    # this function converts a matrix to axis angle representations
    # this matrix is usually a resulting matrix (result of matrix multiplication) in normal use, given as a list
    # returns a list of [rx,ry,rz]
    def convert_matrix_to_axang(matrix1):
        # retrieve values
        a11 = matrix1[0]
        a12 = matrix1[1]
        a13 = matrix1[2]
        a21 = matrix1[3]
        a22 = matrix1[4]
        a23 = matrix1[5]
        a31 = matrix1[6]
        a32 = matrix1[7]
        a33 = matrix1[8]

        # First Half: find the angle
        # find the trace
        # using the formula: trace = a11 + a22 + a33
        trace = a11 + a22 + a33
        # find the angle using the formula: trace(matrix) = 1 + 2 cos(angle)
        angle = acos((trace - 1.0)/2.0)

        # Second Half: calculate the rotation axis
        axisxraw = a32 - a23
        axisyraw = a13 - a31
        axiszraw = a21 - a12
        # normalize axis
        magnitude = sqrt(axisxraw*axisxraw + axisyraw*axisyraw + axiszraw*axiszraw)
        axisxunit = axisxraw / magnitude
        axisyunit = axisyraw / magnitude
        axiszunit = axiszraw / magnitude

        # combine axis and angle into rxryrz representation
        rxout = axisxunit * angle
        ryout = axisyunit * angle
        rzout = axiszunit * angle
        return [rxout, ryout, rzout]
    end

    # this function takes a rotation and calculates the corresponding rotation matrix
    # input is (axis, direction, angle in radians)
    # example is ("x", 1, pi/6) = a 30 degree turn around the x axis in the positive direction (right hand rule)
    # returns a matrix (a list of 9 values)
    def get_rotation_matrix_from_description(axis, direction, angle):
        # get the angle
        a = angle * direction
        # get the axis
        if axis == "x" or axis == "X":
            matrix = [1, 0, 0, 0, cos(a), -1 * sin(a), 0, sin(a), cos(a)]
            return matrix
        end
        if axis == "y" or axis == "Y":
            matrix = [cos(a), 0, sin(a), 0, 1, 0, -1*sin(a), 0, cos(a)]
            return matrix
        end
        if axis == "z" or axis == "Z":
            matrix = [cos(a), -1*sin(a), 0, sin(a), cos(a), 0, 0, 0, 1]
            return matrix
        end
        # bad
        popuptext = "Error in get_rotation_matrix_from_description. "
        # infinite loop
        while 1==1:
          popup(popuptext, title="Code Error",blocking=True)
        end
    end

    def main_calculate_step_right(p11, p12, p21, p22, p3, p13, p23, noncappingsidewallthick, cappingsidewallthick, tcp_pose_top):
        struct1 = analyze_touchpoints_only(p11, p12, p21, p22, p3)
        list1 = analyze_vertical_touchpoints(p11, p12, p13, p21, p22, p23, p3)
        #struct2 = calculate_DOtA_points_right(struct1, list1, chamferover)
        #validity = check_validity_right(struct1, struct2)
        struct2 = calculate_DAaU_step_right(struct1, list1, noncappingsidewallthick, cappingsidewallthick, tcp_pose_top)
        return struct2
    end

    def main_calculate_step_left(p11, p12, p21, p22, p3, p13, p23, noncappingsidewallthick, cappingsidewallthick, tcp_pose_top):
        struct1 = analyze_touchpoints_only(p11, p12, p21, p22, p3)
        list1 = analyze_vertical_touchpoints(p11, p12, p13, p21, p22, p23, p3)
        #struct2 = calculate_DOtA_points_right(struct1, list1, chamferover)
        #validity = check_validity_right(struct1, struct2)
        struct2 = calculate_DAaU_step_left(struct1, list1, cappingsidewallthick, noncappingsidewallthick, tcp_pose_top)
        return struct2
    end

    # analyze_touchpoints_only()
    # it takes 5 arguments as points
    # it returns a struct containing: (pointintersect, heading1, heading2, heading3, l1delxunit, l1delyunit, l2delxunit, l2delyunit)
    #   FIND HEADINGS
    #for each heading, find the angle of the line with respect to the pos x axis. then add/subtract 90 degrees because you want to be perpendicular to that
    # so, heading1 finds the angle (from the +x axis) to the position pointing perpendicularly into the box.
    # we need to be +90 degrees of all 3 headings. (but we can ignore heading 2)
    def step_right_demo(struct1):
        pointintersect = struct1[0]
        x = pointintersect[0]
        y = pointintersect[1]
        z = pointintersect[2]
        heading1 = struct1[1]
        heading1adj1 = heading1 + pi/2 #(90 deg) (parrallel to edge not perpendicular into
        heading1adj2 = heading1adj1 - pi/2 #(90 deg) (from y+ not x+)
        # heading1 == heading1adj2. ok
        m1 = get_rotation_matrix_from_description("z", 1, heading1)
        # at this point we would multiply matrices, but there is only one matrix
        rxryrz = convert_matrix_to_axang(m1)
        point_demo = p[x, y, z, rxryrz[0], rxryrz[1], rxryrz[2]]
        popup(point_demo)
        movej(point_demo, a=1.4, v=0.1)
        popup(point_demo)
        ret = struct(point_demo = point_demo)
        return ret
    end

    # for a right step corner, calculate the toolpath points for a L (under) then Up and Around weld.
    def calculate_LtUA_step_right(struct1, list1, rightwallthick, leftwallthick, tcp_pose_top):
        # get the stuff from the struct
        pointintersect = struct1[0]
        heading1 = struct1[1]
        heading2 = struct1[2]
        heading3 = struct1[3]
        l1delxunit = struct1[4]
        l1delyunit = struct1[5]
        l2delxunit = struct1[6]
        l2delyunit = struct1[7]

        # FIND THE POINTS ON THE LINES OF THE FIRST TURN PATH
        # find locations 8 inches away from  intersect point
        # CONST
        welddistance1 = 3 # first path first leg
        welddistance2 = 3 # first path second leg
        welddistance3 = 8 # vertical weld distance

        # inches
        wd1 = welddistance1 * 25.4 / 1000
        wd2 = welddistance2 * 25.4 / 1000
        wd3 = welddistance3 * 25.4 / 1000
        leftwallthickmm = leftwallthick * 25.4 / 1000 # in this step corner right, this is distance from left edge
        rightwallthickmm =  rightwallthick * 25.4 / 1000 # in this step corner right, this is distance from right edge


        # weld distance is the distance that it will weld. this will make it start at the z height that the user specified
        #wd1 = tcp_pose_top[2] - pointintersect[2] - zup # this will need to change for step corner right

        # point bottom (point of intersection of the two chamfers on the bottom)
        xbottom = pointintersect[0] + l1delxunit * leftwallthickmm + l2delxunit * rightwallthickmm
        ybottom = pointintersect[1] + l1delyunit * leftwallthickmm + l2delyunit * rightwallthickmm
        z = pointintersect[2]

        # point 1
        x = xbottom + l1delxunit * wd1
        y = ybottom + l1delyunit * wd1

        m1 = get_rotation_matrix_from_description("z", 1, heading1)
        # at this point we would multiply matrices, but there is only one matrix
        rxryrz = convert_matrix_to_axang(m1)
        rx = rxryrz[0]
        ry = rxryrz[1]
        rz = rxryrz[2]
        point1 = p[x, y, z, rx, ry, rz]

        # point 2
        point2 = p[xbottom, ybottom, z, rx, ry, rz]

        # point 4
        m1 = get_rotation_matrix_from_description("z", 1, heading3)
        # at this point we would multiply matrices, but there is only one matrix
        rxryrz = convert_matrix_to_axang(m1)
        rx = rxryrz[0]
        ry = rxryrz[1]
        rz = rxryrz[2]
        point4 = p[xbottom, ybottom, z, rx, ry, rz]

        # point 5
        x = xbottom + l2delxunit * wd2
        y = ybottom + l2delyunit * wd2
        point5 = p[x, y, z, rx, ry, rz]


        # form struct
        struct2 = struct(point1=point1, point2=point2, point4=point4, point5=point5, point_1=point1, point_2=point1, point_3=point1, point_4=point1, point_5=point1)
        return struct2
    end

    # step corner with two seams on bottom face
    # vertical seam on left side of corner
    # Down Around and Under weld path, then Back Away
    # the first path uses backofhole TCP, the second path uses pretend_welder TCP
    def calculate_DAaU_step_left(struct1, listleans, rightwallthick, leftwallthick, tcp_pose_top):
        # get the stuff from the struct
        pointintersect = struct1[0]
        heading1 = struct1[1]
        heading2 = struct1[2]
        heading3 = struct1[3]
        l1delxunit = struct1[4]
        l1delyunit = struct1[5]
        l2delxunit = struct1[6]
        l2delyunit = struct1[7]

        # FIND THE POINTS ON THE LINES OF THE FIRST TURN PATH
        # find locations 8 inches away from  intersect point
        # CONST
        welddistance1 = 8 # first path first leg (down)
        welddistance2 = 3 # first path second leg (under) # inches
        welddistance3 = 3 # second path (back away) # inches

        wd1 = tcp_pose_top[2] - pointintersect[2] # the touchpoint minus the corner
        wd2 = welddistance2 * 25.4 / 1000
        wd3 = welddistance3 * 25.4 / 1000
        leftwallthickmm = leftwallthick * 25.4 / 1000 # in this step corner right, this is distance from left edge
        rightwallthickmm =  rightwallthick * 25.4 / 1000 # in this step corner right, this is distance from right edge

        # first, calculate the location of the bottom of the vertical chamfer (where point2 would be if there weren't any circle motion
        x = pointintersect[0] + l2delxunit * rightwallthickmm
        y = pointintersect[1] + l2delyunit * rightwallthickmm
        z = pointintersect[2]
        pointbottomvcham = p[x, y, z, 0, 0, 0]

        # calculate the rxryrz for facing the vertical chamfer, with the preheat down
        rxryrz = convert_heading_to_axang_preheatdown(heading3)
        rx = rxryrz[0]
        ry = rxryrz[1]
        rz = rxryrz[2]

        # next, calculate point1 using the listleans
        point1 = p[x + wd1*listleans[0], y + wd1*listleans[1], z + wd1, rx, ry, rz] # add in the listleans factor to follow the face of the box as we move up

        # calculate rxryrz for point2 and point2a (based on heading1). should be very similar to the heading for point1
        # only use the right side taps for circle move related things
        heading3basedh1 = heading1 - pi/2 # heading1 based on heading3
        rxryrz = convert_heading_to_axang_preheatdown(heading3basedh1)
        rx = rxryrz[0]
        ry = rxryrz[1]
        rz = rxryrz[2]

        # the round over distance is the distance from pointbottomvcham to point2 (which will be the same as distance to p4)
        roundoverdistance = 0.05
        rod = roundoverdistance * 25.4 / 1000
        point2 = p[x, y, z + rod, rx, ry, rz]

        # calculate point2a, which is directly above pointbottomvcham (used to straighten weldpath before circlemove)
        straightlength = 1.0 # the moveP blend radius for the circle move was set to 1.0 mm in FloorCorner. we should be more than 2.0mm away from point2
        sld = straightlength * 25.4 / 1000
        point2a = p[x, y, z + sld, rx, ry, rz]

        # calculate the rxryrz for facing the underneath section, with the preheat facing parallel to the right edge (rx and ry should be 0 because gun is facing up)
        # to convert heading1 into the description, subtract 90 degrees to go parallel  instead of into. subtract 90 degrees to start from y+ instead of x+
        heading1descr = heading1 - pi
        m1 = get_rotation_matrix_from_description("z", 1, heading1descr)
        rxryrz = convert_matrix_to_axang(m1)
        rx = rxryrz[0]
        ry = rxryrz[1]
        rz = rxryrz[2]

        # calculate point4
        p4x = x + l1delxunit * rod
        p4y = y + l1delyunit * rod
        point4 = p[p4x, p4y, z, rx, ry, rz]

        # calculate point5
        p5x = x + l1delxunit * wd2
        p5y = y + l1delyunit * wd2
        point5 = p[p5x, p5y, z, rx, ry, rz]

        # calculate point3
        # we know that the angle is exactly 90 degrees
        delta = calc_rod_midpoint_90deg(rod)
        p3z = z + delta
        p3x = x + delta * l1delxunit
        p3y = y + delta * l1delyunit

        # calculate rxryrz
        m1 = get_rotation_matrix_from_description("x", -1, 45 * pi / 180) # rotation 1: 45 degrees forward about x axis
        m2 = get_rotation_matrix_from_description("z", 1, heading1descr) # rotation 2
        m3 = multiply_matrix(m2, m1) #we rotate m1 first then m2, so we multiply in backwards order: 2 then 1
        rxryrz = convert_matrix_to_axang(m3)
        rx = rxryrz[0]
        ry = rxryrz[1]
        rz = rxryrz[2]
        point3 = p[p3x, p3y, p3z, rx, ry, rz]

        #todo: calculate trail out point

        # calculate back-away (points 201 and 202)
        pushtipforward = 0.006 # 6 millimeters forward. the tip needs to clear the capping wall's angled chamfer to not BONK when getting into position
        p201x = x + l1delxunit * leftwallthickmm + l2delxunit * pushtipforward
        p201y = y + l1delyunit * leftwallthickmm + l2delyunit * pushtipforward

        # calculate rxryrz
        m1 = get_rotation_matrix_from_description("z", 1, heading3)
        # minus pi/2 for the different start point. minus pi/2 for parallel not perpendicular into
        rxryrz = convert_matrix_to_axang(m1)
        rx = rxryrz[0]
        ry = rxryrz[1]
        rz = rxryrz[2]
        point201 = p[p201x, p201y, z, rx, ry, rz]

        # calculate point 202
        p202x = p201x + wd3 * l2delxunit
        p202y = p201y + wd3 * l2delyunit
        point202 = p[p202x, p202y, z, rx, ry, rz]

        struct2 = struct(point1=point1, point2a=point2a, point2=point2, point3=point3, point4=point4, point5=point5, point201=point201, point202=point202)
        return struct2
    end

    # step corner with two seams on bottom face
    # vertical seam on right side of corner
    # Down Around and Under weld path, then Back Away
    # the first path uses backofhole TCP, the second path uses pretend_welder TCP
    def calculate_DAaU_step_right(struct1, listleans, rightwallthick, leftwallthick, tcp_pose_top):
        # get the stuff from the struct
        pointintersect = struct1[0]
        heading1 = struct1[1]
        heading2 = struct1[2]
        heading3 = struct1[3]
        l1delxunit = struct1[4]
        l1delyunit = struct1[5]
        l2delxunit = struct1[6]
        l2delyunit = struct1[7]

        # FIND THE POINTS ON THE LINES OF THE FIRST TURN PATH
        # find locations 8 inches away from  intersect point
        # CONST
        welddistance1 = 8 # first path first leg (down)
        welddistance2 = 3 # first path second leg (under) # inches
        welddistance3 = 3 # second path (back away) # inches

        wd1 = tcp_pose_top[2] - pointintersect[2] # the touchpoint minus the corner
        wd2 = welddistance2 * 25.4 / 1000
        wd3 = welddistance3 * 25.4 / 1000
        leftwallthickmm = leftwallthick * 25.4 / 1000 # in this step corner right, this is distance from left edge
        rightwallthickmm =  rightwallthick * 25.4 / 1000 # in this step corner right, this is distance from right edge

        # first, calculate the location of the bottom of the vertical chamfer (where point2 would be if there weren't any circle motion
        x = pointintersect[0] + l1delxunit * leftwallthickmm
        y = pointintersect[1] + l1delyunit * leftwallthickmm
        z = pointintersect[2]
        pointbottomvcham = p[x, y, z, 0, 0, 0]

        # calculate the rxryrz for facing the vertical chamfer, with the preheat down
        rxryrz = convert_heading_to_axang_preheatdown(heading1)
        rx = rxryrz[0]
        ry = rxryrz[1]
        rz = rxryrz[2]

        # next, calculate point1 using the listleans
        point1 = p[x + wd1*listleans[0], y + wd1*listleans[1], z + wd1, rx, ry, rz] # add in the listleans factor to follow the face of the box as we move up

        # calculate rxryrz for point2 and point2a (based on heading3). should be very similar to the heading for point1
        # only use the left side taps for circle move related things
        heading1basedh3 = heading3 + pi/2 # heading1 based on heading3
        rxryrz = convert_heading_to_axang_preheatdown(heading1basedh3)
        rx = rxryrz[0]
        ry = rxryrz[1]
        rz = rxryrz[2]

        # the round over distance is the distance from pointbottomvcham to point2 (which will be the same as distance to p4)
        roundoverdistance = 0.05
        rod = roundoverdistance * 25.4 / 1000
        point2 = p[x, y, z + rod, rx, ry, rz]

        # calculate point2a, which is directly above pointbottomvcham (used to straighten weldpath before circlemove)
        straightlength = 1.0 # the moveP blend radius for the circle move was set to 1.0 mm in FloorCorner. we should be more than 2.0mm away from point2
        sld = straightlength * 25.4 / 1000
        point2a = p[x, y, z + sld, rx, ry, rz]


        # calculate the rxryrz for facing the underneath section, with the preheat facing parallel to the left edge (rx and ry should be 0 because gun is facing up)
        m1 = get_rotation_matrix_from_description("z", 1, heading3)
        rxryrz = convert_matrix_to_axang(m1)
        rx = rxryrz[0]
        ry = rxryrz[1]
        rz = rxryrz[2]

        # calculate point4
        p4x = x + l2delxunit * rod
        p4y = y + l2delyunit * rod
        point4 = p[p4x, p4y, z, rx, ry, rz]

        # calculate point5
        p5x = x + l2delxunit * wd2
        p5y = y + l2delyunit * wd2
        point5 = p[p5x, p5y, z, rx, ry, rz]

        # calculate point3
        # we know that the angle is exactly 90 degrees
        delta = calc_rod_midpoint_90deg(rod)
        p3z = z + delta
        p3x = x + delta * l2delxunit
        p3y = y + delta * l2delyunit

        # calculate rxryrz
        m1 = get_rotation_matrix_from_description("x", -1, 45 * pi / 180) # rotation 1: 45 degrees forward about x axis
        m2 = get_rotation_matrix_from_description("z", 1, heading3) # rotation 2
        m3 = multiply_matrix(m2, m1) #we rotate m1 first then m2, so we multiply in backwards order: 2 then 1
        rxryrz = convert_matrix_to_axang(m3)
        rx = rxryrz[0]
        ry = rxryrz[1]
        rz = rxryrz[2]
        point3 = p[p3x, p3y, p3z, rx, ry, rz]

        #todo: calculate trail out point

        # calculate back-away (points 201 and 202)
        pushtipforward = 0.006 # 6 millimeters forward. the tip needs to clear the capping wall's angled chamfer to not BONK when getting into position
        p201x = x + l2delxunit * rightwallthickmm + l1delxunit * pushtipforward
        p201y = y + l2delyunit * rightwallthickmm + l1delyunit * pushtipforward

        # calculate rxryrz
        m1 = get_rotation_matrix_from_description("z", 1, heading1 - pi)
        # minus pi/2 for the different start point. minus pi/2 for parallel not perpendicular into
        rxryrz = convert_matrix_to_axang(m1)
        rx = rxryrz[0]
        ry = rxryrz[1]
        rz = rxryrz[2]
        point201 = p[p201x, p201y, z, rx, ry, rz]

        # calculate point 202
        p202x = p201x + wd3 * l1delxunit
        p202y = p201y + wd3 * l1delyunit
        point202 = p[p202x, p202y, z, rx, ry, rz]

        struct2 = struct(point1=point1, point2a=point2a, point2=point2, point3=point3, point4=point4, point5=point5, point201=point201, point202=point202)
        return struct2
    end

    # given a round over distance (in mm), calculate (based on 90 degrees) the distance from corner (line intersection) to midpoint of arc
    # returns a value (in mm) that you need to move from line intersection to midpoint (actual distance will be this times sqrt(2))
    def calc_rod_midpoint_90deg(rod):
        # the factor is (1- 1/sqrt(2))
        factor = 0.292893
        ret = rod * factor
        return ret
    end

    # this is the main entry point for calculations, for Cover Corner.
    # it takes in the 4 touchpoints, analyzes the shape of the box.
    # returns the pathpoints
    # specifically for Around and Down then Straight (AtS)
    # specifically for left-sided boxes (vertical weld on left side of edge)
    def main_calculate_cover(p11, p12, p21, p3, leftwallthick, rightwallthick, leftchoice):
        struct1 = analyze_touchpoints_only_cover(p11, p12, p21, p3)
        if leftchoice:
            struct2 = calculate_AtS_points_cover_left(struct1, leftwallthick, rightwallthick)
        else:
            struct2 = calculate_AtS_points_cover_right(struct1, leftwallthick, rightwallthick)
        end
        #struct2 = calculate_DOtA_points_left_extended(struct1, list1, chamferover, chamferup, tcp_pose_top)
        #struct3 = check_validity_left(struct1, struct2)
        return struct2
    end

    def calculate_AtS_points_cover_left(struct1, leftwallthick, rightwallthick):
        # get the stuff from the struct
        pointintersect = struct1[0]
        heading1 = struct1[1]
        heading2 = struct1[2]
        heading3 = struct1[3]
        l1delxunit = struct1[4]
        l1delyunit = struct1[5]
        l2delxunit = struct1[6]
        l2delyunit = struct1[7]

        # FIND THE POINTS ON THE LINES OF THE FIRST TURN PATH
        # find locations 8 inches away from  intersect point
        # CONST
        welddistance1 = 6 # first path first leg (down)
        welddistance2 = 4 # first path second leg (under) # inches
        welddistance3 = 6 # second path (back away) # inches

        wd1 = welddistance1 * 25.4 / 1000
        wd2 = welddistance2 * 25.4 / 1000
        wd3 = welddistance3 * 25.4 / 1000
        leftwallthickmm = leftwallthick * 25.4 / 1000 # in this step corner right, this is distance from left edge
        rightwallthickmm =  rightwallthick * 25.4 / 1000 # in this step corner right, this is distance from right edge

        # first, check if we need a lift column raise
        # (we do, because for maximum reach we want to make the lift pedestal be even with the top of the covers)
        zpi = pointintersect[2]
        if zpi > 0:
            liftcolumnzneeded = zpi * 1000.0 # the robot uses coordinates in meters, but the lift column uses coordinates in mm
            z = 0
        else:
            z = zpi
        end

        # first, calculate the location of the top of the vertical chamfer (where point2 would be if there weren't any circle motion)
        x = pointintersect[0] + l2delxunit * rightwallthickmm
        y = pointintersect[1] + l2delyunit * rightwallthickmm
        #z = pointintersect[2] # replaced by z of lift column (directly above)
        pointtopvcham = p[x, y, z, 0, 0, 0]

        # calculate the rxryrz for the gun when it's at point1
        # start with rxryrz = 0,0,0 (gun facing up, preheat facing y+ axis.
        # rotate it 180 degrees about x axis. gun facing down, preheat facing y- axis
        # rotate it about 45 degrees ccw about z axis. x+ to heading1 is about 135 degrees. so our angle is heading1 - 90 degrees
        m1 = get_rotation_matrix_from_description("x", -1, 180 * pi / 180) # rotation 1: 180 degrees forward about x axis
        m2 = get_rotation_matrix_from_description("z", 1, heading1 - pi/2) # rotation 2
        m3 = multiply_matrix(m2, m1) #we rotate m1 first then m2, so we multiply in backwards order: 2 then 1
        rxryrz = convert_matrix_to_axang(m3)
        rx = rxryrz[0]
        ry = rxryrz[1]
        rz = rxryrz[2]

        # next, calculate point1
        p1x = x + l1delxunit * wd1
        p1y = y + l1delyunit * wd1
        point1 = p[p1x, p1y, z, rx, ry, rz]

        # the round over distance is the distance from pointbottomvcham to point2 (which will be the same as distance to p4)
        roundoverdistance = 0.05
        rod = roundoverdistance * 25.4 / 1000
        p2x = x + l1delxunit * rod
        p2y = y + l1delyunit * rod
        point2 = p[p2x, p2y, z, rx, ry, rz]

        # make point2a, colinear between p1 and p2, which will be the place the welder shuts off during motion
        wtod = 0.015 # weldturnoffdistance # meters from pointtopvcham # 10 mm (1.0 seconds)
        p2ax = x + l1delxunit * wtod
        p2ay = y + l1delyunit * wtod
        point2a = p[p2ax, p2ay, z, rx, ry, rz]

        # calculate the rxryrz for facing the down the left side of the box
        # rotate about x 90 (forward). then rotate about z ~ 45 (ccw)
        m1 = get_rotation_matrix_from_description("x", -1, 90 * pi / 180)
        m2 = get_rotation_matrix_from_description("z", 1, heading1 - pi/2)
        m3 = multiply_matrix(m2, m1) #we rotate m1 first then m2, so we multiply in backwards order: 2 then 1
        rxryrz = convert_matrix_to_axang(m3)
        rx = rxryrz[0]
        ry = rxryrz[1]
        rz = rxryrz[2]

        # calculate point4
        point4 = p[x, y, z - rod, rx, ry, rz]

        # calculate point5
        point5 = p[x, y, z - wd2, rx, ry, rz]

        # calculate point3
        # we know that the angle is exactly 90 degrees
        delta = calc_rod_midpoint_90deg(rod)
        p3z = z - delta
        p3x = x + delta * l1delxunit
        p3y = y + delta * l1delyunit

        # calculate rxryrz
        m1 = get_rotation_matrix_from_description("x", -1, 135 * pi / 180) # rotation 1: 135 degrees forward about x axis
        m2 = get_rotation_matrix_from_description("z", 1, heading1 - pi/2)
        m3 = multiply_matrix(m2, m1) #we rotate m1 first then m2, so we multiply in backwards order: 2 then 1
        rxryrz = convert_matrix_to_axang(m3)
        rx = rxryrz[0]
        ry = rxryrz[1]
        rz = rxryrz[2]
        point3 = p[p3x, p3y, p3z, rx, ry, rz]

        #todo: calculate trail out point

        # calculate back-away (points 201 and 202)
        pushtipforward = 0.006 # 6 millimeters forward. the tip needs to clear the capping wall's angled chamfer to not BONK when getting into position
        p201x = x + l1delxunit * leftwallthickmm + l2delxunit * pushtipforward
        p201y = y + l1delyunit * leftwallthickmm + l2delyunit * pushtipforward

        # calculate rxryrz
        # rotate 180 degrees about x. then rotate (90 deg + heading3 degrees) about z ccw
        m1 = get_rotation_matrix_from_description("x", -1, 180 * pi / 180)
        m2 = get_rotation_matrix_from_description("z", 1, heading3 + pi/2)
        m3 = multiply_matrix(m2, m1) #we rotate m1 first then m2, so we multiply in backwards order: 2 then 1
        rxryrz = convert_matrix_to_axang(m3)
        rx = rxryrz[0]
        ry = rxryrz[1]
        rz = rxryrz[2]
        point201 = p[p201x, p201y, z, rx, ry, rz]

        # calculate point 201's preheat
        pushtipforward2 = 0.012 - pushtipforward # 12 mm forward to clear the existing extrudant (but still have the extrudant from this extrusion join the existing). subtract from previous to make it constant even if you change pushtipforward1
        preheatdistance = 0.010 # 10 mm . above what it would be pushed down
        point201a = p[p201x, p201y, z + preheatdistance, rx, ry, rz]
        p201bx = p201x + l2delxunit * pushtipforward2
        p201by = p201y + l2delyunit * pushtipforward2
        point201b = p[p201bx, p201by, z + preheatdistance, rx, ry, rz]
        point201c = p[p201bx, p201by, z, rx, ry, rz]

        # calculate point 202
        p202x = p201x + wd3 * l2delxunit
        p202y = p201y + wd3 * l2delyunit
        point202 = p[p202x, p202y, z, rx, ry, rz]

        struct2 = struct(point1=point1, point2=point2, point3=point3, point4=point4, point5=point5, point201=point201, point202=point202, point201a=point201a, point201b=point201b, point201c=point201c, point2a=point2a)
        return struct2
    end

    def calculate_AtS_points_cover_right(struct1, leftwallthick, rightwallthick):
        # get the stuff from the struct
        pointintersect = struct1[0]
        heading1 = struct1[1]
        heading2 = struct1[2]
        heading3 = struct1[3]
        l1delxunit = struct1[4]
        l1delyunit = struct1[5]
        l2delxunit = struct1[6]
        l2delyunit = struct1[7]

        # FIND THE POINTS ON THE LINES OF THE FIRST TURN PATH
        # find locations 8 inches away from  intersect point
        # CONST
        welddistance1 = 6 # first path first leg (down)
        welddistance2 = 4 # first path second leg (under) # inches
        welddistance3 = 6 # second path (back away) # inches

        wd1 = welddistance1 * 25.4 / 1000
        wd2 = welddistance2 * 25.4 / 1000
        wd3 = welddistance3 * 25.4 / 1000
        leftwallthickmm = leftwallthick * 25.4 / 1000 # in this step corner right, this is distance from left edge
        rightwallthickmm =  rightwallthick * 25.4 / 1000 # in this step corner right, this is distance from right edge

        # first, check if we need a lift column raise
        # (we do, because for maximum reach we want to make the lift pedestal be even with the top of the covers)
        zpi = pointintersect[2]
        if zpi > 0:
            liftcolumnzneeded = zpi * 1000.0 # the robot uses coordinates in meters, but the lift column uses coordinates in mm
            z = 0
        else:
            z = zpi
        end

        # first, calculate the location of the top of the vertical chamfer (where point2 would be if there weren't any circle motion)
        x = pointintersect[0] + l1delxunit * leftwallthickmm
        y = pointintersect[1] + l1delyunit * leftwallthickmm
        #z = pointintersect[2] # replaced by z of lift column (directly above)
        pointtopvcham = p[x, y, z, 0, 0, 0]

        # calculate the rxryrz for the gun when it's at point1
        # start with rxryrz = 0,0,0 (gun facing up, preheat facing y+ axis.
        # rotate it 180 degrees about x axis. gun facing down, preheat facing y- axis
        # rotate it about 135 degrees ccw about z axis. x+ to heading3 is about 225 degrees. so our angle is heading3 - 90 degrees
        m1 = get_rotation_matrix_from_description("x", -1, 180 * pi / 180) # rotation 1: 180 degrees forward about x axis
        m2 = get_rotation_matrix_from_description("z", 1, heading3 - pi/2) # rotation 2
        m3 = multiply_matrix(m2, m1) #we rotate m1 first then m2, so we multiply in backwards order: 2 then 1
        rxryrz = convert_matrix_to_axang(m3)
        rx = rxryrz[0]
        ry = rxryrz[1]
        rz = rxryrz[2]

        # next, calculate point1
        p1x = x + l2delxunit * wd1
        p1y = y + l2delyunit * wd1
        point1 = p[p1x, p1y, z, rx, ry, rz]

        # the round over distance is the distance from pointbottomvcham to point2 (which will be the same as distance to p4)
        roundoverdistance = 0.05
        rod = roundoverdistance * 25.4 / 1000
        p2x = x + l2delxunit * rod
        p2y = y + l2delyunit * rod
        point2 = p[p2x, p2y, z, rx, ry, rz]

        # make point2a, colinear between p1 and p2, which will be the place the welder shuts off during motion
        wtod = 0.015 # weldturnoffdistance # meters from pointtopvcham # 10 mm (1.0 seconds)
        p2ax = x + l2delxunit * wtod
        p2ay = y + l2delyunit * wtod
        point2a = p[p2ax, p2ay, z, rx, ry, rz]

        # calculate the rxryrz for facing the down the right side of the box
        # rotate about x 90 (forward). then rotate about z ~ 135 (ccw)
        m1 = get_rotation_matrix_from_description("x", -1, 90 * pi / 180)
        m2 = get_rotation_matrix_from_description("z", 1, heading3 - pi/2)
        m3 = multiply_matrix(m2, m1) #we rotate m1 first then m2, so we multiply in backwards order: 2 then 1
        rxryrz = convert_matrix_to_axang(m3)
        rx = rxryrz[0]
        ry = rxryrz[1]
        rz = rxryrz[2]

        # calculate point4
        point4 = p[x, y, z - rod, rx, ry, rz]

        # calculate point5
        point5 = p[x, y, z - wd2, rx, ry, rz]

        # calculate point3
        # we know that the angle is exactly 90 degrees
        delta = calc_rod_midpoint_90deg(rod)
        p3z = z - delta
        p3x = x + delta * l2delxunit
        p3y = y + delta * l2delyunit

        # calculate rxryrz
        m1 = get_rotation_matrix_from_description("x", -1, 135 * pi / 180) # rotation 1: 135 degrees forward about x axis
        m2 = get_rotation_matrix_from_description("z", 1, heading3 - pi/2)
        m3 = multiply_matrix(m2, m1) #we rotate m1 first then m2, so we multiply in backwards order: 2 then 1
        rxryrz = convert_matrix_to_axang(m3)
        rx = rxryrz[0]
        ry = rxryrz[1]
        rz = rxryrz[2]
        point3 = p[p3x, p3y, p3z, rx, ry, rz]

        #todo: calculate trail out point

        # calculate back-away (points 201 and 202)
        pushtipforward = 0.006 # 6 millimeters forward. the tip needs to clear the capping wall's angled chamfer to not BONK when getting into position
        p201x = x + l2delxunit * rightwallthickmm + l1delxunit * pushtipforward
        p201y = y + l2delyunit * rightwallthickmm + l1delyunit * pushtipforward

        # calculate rxryrz
        # rotate 180 degrees about x. then rotate (90 deg + heading1 degrees) about z ccw
        m1 = get_rotation_matrix_from_description("x", -1, 180 * pi / 180)
        m2 = get_rotation_matrix_from_description("z", 1, heading1 + pi/2)
        m3 = multiply_matrix(m2, m1) #we rotate m1 first then m2, so we multiply in backwards order: 2 then 1
        rxryrz = convert_matrix_to_axang(m3)
        rx = rxryrz[0]
        ry = rxryrz[1]
        rz = rxryrz[2]
        point201 = p[p201x, p201y, z, rx, ry, rz]

        # calculate point 201's preheat
        pushtipforward2 = 0.012 - pushtipforward # 12 mm forward to clear the existing extrudant (but still have the extrudant from this extrusion join the existing). subtract from previous to make it constant even if you change pushtipforward1
        preheatdistance = 0.010 # 10 mm . above what it would be pushed down
        point201a = p[p201x, p201y, z + preheatdistance, rx, ry, rz]
        p201bx = p201x + l1delxunit * pushtipforward2
        p201by = p201y + l1delyunit * pushtipforward2
        point201b = p[p201bx, p201by, z + preheatdistance, rx, ry, rz]
        point201c = p[p201bx, p201by, z, rx, ry, rz]

        # calculate point 202
        p202x = p201x + wd3 * l1delxunit
        p202y = p201y + wd3 * l1delyunit
        point202 = p[p202x, p202y, z, rx, ry, rz]

        struct2 = struct(point1=point1, point2=point2, point3=point3, point4=point4, point5=point5, point201=point201, point202=point202, point201a=point201a, point201b=point201b, point201c=point201c, point2a=point2a)
        return struct2
    end

    def main_calculate_cover_straight(p11, p12, p21, p22, sidewallthick, leftpoint, rightpoint):
        struct1 = analyze_touchpoints_only_cover_straight(p11, p12, p21, p22, leftpoint)
        struct2 = calculate_straight_points_cover(struct1, sidewallthick, leftpoint, rightpoint)
        #struct2 = calculate_DOtA_points_left_extended(struct1, list1, chamferover, chamferup, tcp_pose_top)
        #struct3 = check_validity_left(struct1, struct2)
        return struct2

    end

    # calculates the line of intersection of the sidewall plane (assumed vertical) and the cover plane (assumed perpendicular to sidewall plane)
    # returns a struct containing point0 (point on the intersection line, same y as leftpoint) and 3 components of the unit vector left to right and 2 components of the other direction in 2d
    def analyze_touchpoints_only_cover_straight(p11, p12, p21, p22, leftpoint):
        # calculate slope of sidewall in x-y plane
        # get the raw points from the first line
        l1p1x=p11[0]
        l1p1y=p11[1]
        l1p2x=p12[0]
        l1p2y=p12[1]

        # equate the first line in 2d space
        ml1 = (l1p2y-l1p1y) / (l1p2x-l1p1x)

        # b = y - mx
        bl1 = l1p1y - ml1 * l1p1x

        # calculate the cover plane
        # if two planes are perpendicular, then their normal vectors must be perpendicular.
        # the first planes normal vector is n1, which is taken from the equation of the plane ax + by + cz = d -> <a, b, c>
        # the second plane's normal vector is perpendicular to all vectors contained in the plane
        # p21 to p22 is a vector v contained within plane 2.
        # n2 is normal to both n1 AND v. to achieve a vector that is normal to both, take the cross product

        # plane 1 (y = mx + b) -> (b = -mx +1y +0z)
        n1 = [-1 * ml1, 1, 0]

        # v=P2−P1=(x2−x1,y2−y1,z2−z1)
        v = [p21[0]-p22[0], p21[1]-p22[1], p21[2]-p22[2]]

        #v n2 = cross product of n1 and v
        n2x = n1[1]*v[2] - n1[2]*v[1]
        n2y = n1[2]*v[0] - n1[0]*v[2]
        n2z = n1[0]*v[1] - n1[1]*v[0]
        n2 = [n2x, n2y, n2z]

        # find the d of the second plane
        # n2x * x + n2y * y + n2z * z = d0
        d = n2x * p21[0] + n2y * p21[1] + n2z * p21[2]

        # find the intersection line of the two planes
        # find the direction vector of that line by taking the cross product of the normal vector of those two planes
        v3x = n1[1]*n2[2] - n1[2]*n2[1]
        v3y = n1[2]*n2[0] - n1[0]*n2[2]
        v3z = n1[0]*n2[1] - n1[1]*n2[0]
        v3 = [v3x, v3y, v3z]

        # normalize the vector so the magnitude is 1
        magnitude2 = v3x * v3x + v3y * v3y + v3z * v3z
        magnitude = sqrt(magnitude2)
        v3xunit = v3x/magnitude
        v3yunit = v3y/magnitude
        v3zunit = v3z/magnitude

        # make sure it is going the right way (from left to right). make sure the v3yunit is positive
        if v3yunit < 0:
            v3xunit = v3xunit * -1
            v3yunit = v3yunit * -1
            v3zunit = v3zunit * -1
        end

        # next we have to find a point on the line by setting one of the dimensions and solving the system of equations
        # i will pick the y value of the left teach point
        y = leftpoint[1]
        # plane 1: -ml1 * x + 1 * y + 0 * z = bl1
        # -ml1 * x = bl1 - y
        x = (bl1 - y)/ (-1 * ml1)
        # plane 2: d = n2x * x + n2y * y + n2z * z
        # (d - n2x * x - n2y * y) = n2z * z
        z = (d - n2x * x - n2y * y) / n2z

        # make point0 into a pose
        point0 = p[x, y, z, 0, 0, 0]

        # find heading of main line
        heading1 = convert_uv_to_heading(v3xunit, v3yunit)

        # make a unit vector perpendicular to this one in the xy plane pointing x -. will be used to move over the chamfer distance
        ml2 = -1 / ml1
        # y = ml2 * x + unknownB
        # vector = [1, ml2]
        mag2 = 1 + ml2 * ml2
        mag = sqrt(mag2)
        v4xunit = 1 / mag
        v4yunit = ml2 / mag
        # switch is to the x direction is negative
        v4xunit = -1 * v4xunit
        v4yunit = -1 * v4yunit

        ret = struct(point0=point0, v3xunit=v3xunit, v3yunit=v3yunit, v3zunit=v3zunit, heading1=heading1, v4xunit=v4xunit, v4yunit=v4yunit)
        return ret
    end

    def calculate_straight_points_cover(struct1, sidewallthick, leftpointteach, rightpointteach):
        # get the stuff
        point0 = struct1[0]
        p0x = point0[0]
        p0y = point0[1]
        p0z = point0[2]
        v3xunit = struct1[1]
        v3yunit = struct1[2]
        v3zunit = struct1[3]
        heading1 = struct1[4]
        v4xunit = struct1[5]
        v4yunit = struct1[6]
        sidewallthick = sidewallthick
        lpy = leftpointteach[1]
        rpy = rightpointteach[1]

        # first, check if we need a lift column raise
        # (we do, because for maximum reach we want to make the lift pedestal be even with the top of the covers)
        zpi = p0z
        if zpi > 0:
            liftcolumnzneeded = zpi * 1000.0 # the robot uses coordinates in meters, but the lift column uses coordinates in mm
            coverz = 0
        else:
            coverz = zpi
        end

        # calculate pointtopvcham
        chamferover = sidewallthick * 25.4 / 1000.0
        tiltraise = 0.006 # 6 mm raise needed for the tip to clear the plane during tiltback
        x = p0x + v4xunit * chamferover
        y = p0y + v4yunit * chamferover
        z = coverz + tiltraise

        # calculate rxryrz for tilted back
        # 3 rotations to make this happen.
        # start point is straight up with the preheat pointed in the +y direction.
        # first rotation is 180 degrees about x direction. gun is now pointing straight down with preheat facing -y direction
        m1 = get_rotation_matrix_from_description("x", 1, 180 * pi / 180)
        # second rotation is a 10 degree turn about the x axis (negative direction)
        m2 = get_rotation_matrix_from_description("x", -1, 10 * pi / 180)
        # third rotation is about 180 degrees about the z axis. starting from the -y axis, go until you get to heading1. that will equal heading1 plus 90 degrees
        m3 = get_rotation_matrix_from_description("z", 1, pi/2 + heading1)
        # combine them by multiplying m3 * m2 * m1
        # matrix multiplication is not commutative but it IS associative, so you can do this whichever order
        m4 = multiply_matrix(m2, m1)
        m5 = multiply_matrix(m3, m4)
        rxryrzt = convert_matrix_to_axang(m5)
        rxt = rxryrzt[0]
        ryt = rxryrzt[1]
        rzt = rxryrzt[2]
        pointtopvcham = p[x, y, z, rxt, ryt, rzt]

        # calculate point1 (preheat)
        dist = -1 * 25.4 / 1000.0 # move back 1 inch from
        p1x = x + dist * v3xunit
        p1y = y + dist * v3yunit
        p1z = z + dist * v3zunit
        point1 = p[p1x, p1y, p1z, rxt, ryt, rzt]

        # calculate point2 (start of flatten)
        dist = 0.5 * 25.4 / 1000.0  # half an inch past the top of v chamfer
        p2x = x + dist * v3xunit
        p2y = y + dist * v3yunit
        p2z = z + dist * v3zunit
        point2 = p[p2x, p2y, p2z, rxt, ryt, rzt]

        # calculate rxryrz for nontilted
        # first rotation is 180 degrees about x direction. gun is now pointing straight down with preheat facing -y direction
        m1 = get_rotation_matrix_from_description("x", 1, 180 * pi / 180)
        # third rotation is about 180 degrees about the z axis. starting from the -y axis, go until you get to heading1. that will equal heading1 plus 90 degrees
        m3 = get_rotation_matrix_from_description("z", 1, pi/2 + heading1)
        m5 = multiply_matrix(m3, m1)
        rxryrz = convert_matrix_to_axang(m5)
        rx = rxryrz[0]
        ry = rxryrz[1]
        rz = rxryrz[2]

        # calculate point3 (end of flatten)
        dist = 1.5 * 25.4 / 1000.0  # 1.5 inches past top of v chamfer
        p3x = x + dist * v3xunit
        p3y = y + dist * v3yunit
        p3z = coverz + dist * v3zunit
        point3 = p[p3x, p3y, p3z, rx, ry, rz]

        # calculate distance between leftpoint and rightpoint
        # we have the y distance. we need to find the total distance.
        # the unit vector (v3) should have a magnitude of 1. that's what analyze_touchpoints_only_cover_straight() calculated.
        # so the total distance is y distance * 1 / v3yunit
        ydist = rpy - lpy
        totdist = ydist / v3yunit

        # calculate pointtopvcham2
        x2 = x + v3xunit * totdist
        y2 = y + v3yunit * totdist
        z2 = z + v3zunit * totdist

        # calculate point4 (start of unflatten)
        dist = -1.5 * 25.4 / 1000.0
        p4x = x2 + v3xunit * dist
        p4y = y2 + v3yunit * dist
        p4z = z2 + v3zunit * dist - tiltraise
        point4 = p[p4x, p4y, p4z, rx, ry, rz]

        # calculate point5 (end of unflatten)
        dist = -0.5 * 25.4 / 1000.0
        p5x = x2 + v3xunit * dist
        p5y = y2 + v3yunit * dist
        p5z = z2 + v3zunit * dist
        point5 = p[p5x, p5y, p5z, rxt, ryt, rzt]

        # calculate point6 (end of smear)
        dist = 2 * 25.4 / 1000.0
        p6x = x2 + v3xunit * dist
        p6y = y2 + v3yunit * dist
        p6z = z2 + v3zunit * dist
        point6 = p[p6x, p6y, p6z, rxt, ryt, rzt]


        # return struct
        ret = struct(pointtopvcham=pointtopvcham, point1=point1, point2=point2, point3=point3, point4=point4, point5=point5, point6=point6)
        return ret


    end

    def main_calculate_floor_straight(p11, p12, p21, p22, floorthick, leftpoint, rightpoint):
        struct1 = analyze_touchpoints_only_cover_straight(p11, p12, p21, p22, leftpoint)
        struct2 = calculate_straight_points_floor(struct1, floorthick, leftpoint, rightpoint)
        #struct2 = calculate_DOtA_points_left_extended(struct1, list1, chamferover, chamferup, tcp_pose_top)
        #struct3 = check_validity_left(struct1, struct2)
        return struct2

    end

    # the path for welding a floor straight weld with v chisels on both sides.
    # start at the right side and move left.
    def calculate_straight_points_floor(struct1, floorthick, leftpointteach, rightpointteach):
        # get the stuff
        point0 = struct1[0]
        p0x = point0[0]
        p0y = point0[1]
        p0z = point0[2]
        v3xunit = struct1[1]
        v3yunit = struct1[2]
        v3zunit = struct1[3]
        heading1 = struct1[4]
        v4xunit = struct1[5]
        v4yunit = struct1[6]
        lpy = leftpointteach[1]
        rpy = rightpointteach[1]

        # first, check if we need a lift column raise
        # (we do not, because the floors are low)
        zpi = p0z
        floorz = zpi

        # calculate pointtopvcham (left point) (tilted and tiltraised)
        chamferup = floorthick * 25.4 / 1000.0
        tiltraise = 0.006 # 6 mm raise needed for the tip to clear the plane during tiltback
        # on this one, move the tiltraise distance sideways (towards robot) and the chamferover distance up
        x = p0x + v4xunit * tiltraise * -1
        y = p0y + v4yunit * tiltraise * -1
        z = floorz + chamferup

        # calculate rxryrz for tilted back
        # 3 rotations to make this happen.
        # start point is straight up with the preheat pointed in the +y direction.
        # first rotation is 90 degrees about y axis. positive direction. gun is now pointing in the x+ direction with preheat facing +y direction
        m1 = get_rotation_matrix_from_description("y", 1, 90 * pi / 180)
        # second rotation is about 180 degrees about the z axis. heading1 plus 90 degrees. gun is now pointing directly into the sidewall
        m2 = get_rotation_matrix_from_description("z", 1, pi/2 + heading1)
        # third rotation is 10 degrees about the z axis. gun is now tilted back 10 degrees from the sidewall
        m3 = get_rotation_matrix_from_description("z", 1, 10 * pi / 180)
        # combine them by multiplying m3 * m2 * m1
        # matrix multiplication is not commutative but it IS associative, so you can do this whichever order
        m4 = multiply_matrix(m2, m1)
        m5 = multiply_matrix(m3, m4)
        rxryrzt = convert_matrix_to_axang(m5)
        rxt = rxryrzt[0]
        ryt = rxryrzt[1]
        rzt = rxryrzt[2]
        # the non tilted angle is just m4
        rxryrz = convert_matrix_to_axang(m4)
        rx = rxryrz[0]
        ry = rxryrz[1]
        rz = rxryrz[2]
        pointtopvcham = p[x, y, z, rxt, ryt, rzt]

        # calculate distance between leftpoint and rightpoint
        # we have the y distance. we need to find the total distance.
        # the unit vector (v3) should have a magnitude of 1. that's what analyze_touchpoints_only_cover_straight() calculated.
        # so the total distance is y distance * 1 / v3yunit
        ydist = rpy - lpy
        totdist = ydist / v3yunit

        # calculate pointtopvcham2 (right point) (tilted and tiltraised)
        x2 = x + v3xunit * totdist
        y2 = y + v3yunit * totdist
        z2 = z + v3zunit * totdist
        pointtopvcham2 = p[x2, y2, z2, rxt, ryt, rzt]

        # calculate point1 (preheat)
        dist = 1 * 25.4 / 1000.0 # move back 1 inch from ptvc2 (in this case back means positive)
        p1x = x2 + dist * v3xunit
        p1y = y2 + dist * v3yunit
        p1z = z2 + dist * v3zunit
        point1 = p[p1x, p1y, p1z, rxt, ryt, rzt]

        # calculate point2 (start of flatten)
        dist = -0.5 * 25.4 / 1000.0  # half an inch past the top of v chamfer
        p2x = x2 + dist * v3xunit
        p2y = y2 + dist * v3yunit
        p2z = z2 + dist * v3zunit
        point2 = p[p2x, p2y, p2z, rxt, ryt, rzt]

        # calculate point3 (end of flatten)
        dist = -1.5 * 25.4 / 1000.0  # 1.5 inches past top of v chamfer
        p3x = x2 + dist * v3xunit + tiltraise * v4xunit
        p3y = y2 + dist * v3yunit + tiltraise * v4yunit
        p3z = z2 + dist * v3zunit
        point3 = p[p3x, p3y, p3z, rx, ry, rz]

        # calculate point4 (start of unflatten)
        dist = 1.5 * 25.4 / 1000.0
        p4x = x + v3xunit * dist + tiltraise * v4xunit
        p4y = y + v3yunit * dist + tiltraise * v4yunit
        p4z = z + v3zunit * dist
        point4 = p[p4x, p4y, p4z, rx, ry, rz]

        # calculate point5 (end of unflatten)
        dist = 0.5 * 25.4 / 1000.0
        p5x = x + v3xunit * dist
        p5y = y + v3yunit * dist
        p5z = z + v3zunit * dist
        point5 = p[p5x, p5y, p5z, rxt, ryt, rzt]

        # calculate point6 (end of smear)
        dist = -2 * 25.4 / 1000.0
        p6x = x + v3xunit * dist
        p6y = y + v3yunit * dist
        p6z = z + v3zunit * dist
        point6 = p[p6x, p6y, p6z, rxt, ryt, rzt]

        # return struct
        ret = struct(pointtopvcham=pointtopvcham, point1=point1, point2=point2, point3=point3, point4=point4, point5=point5, point6=point6)
        return ret

    end
    $ 286 "path_pre≔get_straight_homing_pathpoints_floor(tcp_pose_left,tcp_pose_right)"
    global path_pre=get_straight_homing_pathpoints_floor(tcp_pose_left,tcp_pose_right)
    $ 287 "ph1≔path_pre[0]"
    global ph1=path_pre[0]
    $ 288 "ph2≔path_pre[1]"
    global ph2=path_pre[1]
    $ 289 "ph3≔path_pre[2]"
    global ph3=path_pre[2]
    $ 290 "ph4≔path_pre[3]"
    global ph4=path_pre[3]
    $ 291 "ph4a≔p[ph4[0]+0.1,ph4[1],ph4[2],ph4[3],ph4[4],ph4[5]]"
    global ph4a=p[ph4[0]+0.1,ph4[1],ph4[2],ph4[3],ph4[4],ph4[5]]
    $ 292 "MoveL"
    $ 293 "Direction: Base X+"
    global move_thread_flag_293=0
    thread move_thread_293():
      enter_critical
      move_thread_flag_293 = 1
      local towardsPos=calculate_point_to_move_towards(p[0.0,0.0,0.0,0.0,0.0,0.0], [1.0,0.0,0.0], 0.1)
      movel(towardsPos, a=1.2, v=0.25)
      move_thread_flag_293 = 2
      exit_critical
    end
    move_thread_flag_293 = 0
    move_thread_han_293 = run move_thread_293()
    while (True):
      sleep(1.0E-10)
      if (move_thread_flag_293 > 1):
        join move_thread_han_293
        $ 294 "Until (distance)"
        break
      end
      sync()
    end
    $ 295 "MoveJ"
    $ 297 "Waypoint_1" "breakAfter"
    movej(get_inverse_kin(Waypoint_1_p, qnear=Waypoint_1_q), a=1.3962634015954636, v=1.0471975511965976)
    $ 298 "MoveL"
    $ 299 "ph1" "breakAfter"
    movel(ph1, a=0.2, v=0.25)
    $ 300 "MoveL"
    $ 301 "Direction: Base X-"
    global move_thread_flag_301=0
    thread move_thread_301():
      enter_critical
      move_thread_flag_301 = 1
      local towardsPos=calculate_point_to_move_towards(p[0.0,0.0,0.0,0.0,0.0,0.0], [-1.0,0.0,0.0], 1000.0)
      movel(towardsPos, a=0.1, v=0.02)
      move_thread_flag_301 = 2
      exit_critical
    end
    move_thread_flag_301 = 0
    move_thread_han_301 = run move_thread_301()
    while (True):
      local targetTcpDirection=get_target_tcp_speed()
      local stepsToRetract=tool_contact(direction=targetTcpDirection)
      if (stepsToRetract > 0):
        kill move_thread_han_301
        stopl(3.0)
        local backTrackMovement=get_actual_joint_positions_history(stepsToRetract)
        local contactPose=get_forward_kin(backTrackMovement)
        local posDir=[targetTcpDirection[0],targetTcpDirection[1],targetTcpDirection[2]]
        local retractTo=contactPose
        if (norm(posDir) > 1e-6):
          local normalizedPosDir=normalize(posDir)
          local additionalRetraction=p[normalizedPosDir[0] * 0.0, normalizedPosDir[1] * 0.0, normalizedPosDir[2] * 0.0, 0, 0, 0]
          retractTo = pose_sub(contactPose, additionalRetraction)
        end
        movel(retractTo, a=3.0, v=0.1)
        $ 302 "Until (tool_contact_detection)"
        break
      end
      sync()
    end
    $ 303 "p11≔get_actual_tcp_pose()"
    global p11= get_actual_tcp_pose ()
    $ 304 "MoveL"
    $ 305 "ph1" "breakAfter"
    movel(ph1, a=1.2, v=0.25)
    $ 306 "ph2" "breakAfter"
    movel(ph2, a=1.2, v=0.25)
    $ 307 "MoveL"
    $ 308 "Direction: Base X-"
    global move_thread_flag_308=0
    thread move_thread_308():
      enter_critical
      move_thread_flag_308 = 1
      local towardsPos=calculate_point_to_move_towards(p[0.0,0.0,0.0,0.0,0.0,0.0], [-1.0,0.0,0.0], 1000.0)
      movel(towardsPos, a=0.1, v=0.02)
      move_thread_flag_308 = 2
      exit_critical
    end
    move_thread_flag_308 = 0
    move_thread_han_308 = run move_thread_308()
    while (True):
      local targetTcpDirection=get_target_tcp_speed()
      local stepsToRetract=tool_contact(direction=targetTcpDirection)
      if (stepsToRetract > 0):
        kill move_thread_han_308
        stopl(3.0)
        local backTrackMovement=get_actual_joint_positions_history(stepsToRetract)
        local contactPose=get_forward_kin(backTrackMovement)
        local posDir=[targetTcpDirection[0],targetTcpDirection[1],targetTcpDirection[2]]
        local retractTo=contactPose
        if (norm(posDir) > 1e-6):
          local normalizedPosDir=normalize(posDir)
          local additionalRetraction=p[normalizedPosDir[0] * 0.0, normalizedPosDir[1] * 0.0, normalizedPosDir[2] * 0.0, 0, 0, 0]
          retractTo = pose_sub(contactPose, additionalRetraction)
        end
        movel(retractTo, a=3.0, v=0.1)
        $ 309 "Until (tool_contact_detection)"
        break
      end
      sync()
    end
    $ 317 "p12≔get_actual_tcp_pose()"
    global p12= get_actual_tcp_pose ()
    $ 318 "MoveJ"
    $ 319 "ph2" "breakAfter"
    movej(ph2, a=1.3962634015954636, v=1.0471975511965976)
    $ 320 "MoveL"
    $ 321 "ph1" "breakAfter"
    movel(ph1, a=1.2, v=0.25)
    $ 322 "MoveJ"
    $ 324 "Waypoint_3" "breakAfter"
    movej(get_inverse_kin(Waypoint_3_p, qnear=Waypoint_3_q), a=1.3962634015954636, v=1.0471975511965976)
    $ 332 "Waypoint_17" "breakAfter"
    movej(get_inverse_kin(Waypoint_17_p, qnear=Waypoint_17_q), a=1.3962634015954636, v=1.0471975511965976)
    $ 333 "Waypoint_16" "breakAfter"
    movej(get_inverse_kin(Waypoint_16_p, qnear=Waypoint_16_q), a=1.3962634015954636, v=1.0471975511965976)
    $ 339 "MoveL"
    $ 340 "ph4a" "breakAfter"
    movel(ph4a, a=1.2, v=0.25)
    $ 341 "ph3" "breakAfter"
    movel(ph3, a=1.2, v=0.25)
    $ 342 "MoveL"
    $ 343 "Direction: Base Z+"
    global move_thread_flag_343=0
    thread move_thread_343():
      enter_critical
      move_thread_flag_343 = 1
      local towardsPos=calculate_point_to_move_towards(p[0.0,0.0,0.0,0.0,0.0,0.0], [0.0,0.0,1.0], 1000.0)
      movel(towardsPos, a=0.1, v=0.02)
      move_thread_flag_343 = 2
      exit_critical
    end
    move_thread_flag_343 = 0
    move_thread_han_343 = run move_thread_343()
    while (True):
      local targetTcpDirection=get_target_tcp_speed()
      local stepsToRetract=tool_contact(direction=targetTcpDirection)
      if (stepsToRetract > 0):
        kill move_thread_han_343
        stopl(3.0)
        local backTrackMovement=get_actual_joint_positions_history(stepsToRetract)
        local contactPose=get_forward_kin(backTrackMovement)
        local posDir=[targetTcpDirection[0],targetTcpDirection[1],targetTcpDirection[2]]
        local retractTo=contactPose
        if (norm(posDir) > 1e-6):
          local normalizedPosDir=normalize(posDir)
          local additionalRetraction=p[normalizedPosDir[0] * 0.0, normalizedPosDir[1] * 0.0, normalizedPosDir[2] * 0.0, 0, 0, 0]
          retractTo = pose_sub(contactPose, additionalRetraction)
        end
        movel(retractTo, a=3.0, v=0.1)
        $ 344 "Until (tool_contact_detection)"
        break
      end
      sync()
    end
    $ 345 "p21≔get_actual_tcp_pose()"
    global p21= get_actual_tcp_pose ()
    $ 346 "MoveL"
    $ 347 "ph3" "breakAfter"
    movel(ph3, a=1.2, v=0.25)
    $ 348 "MoveL"
    $ 349 "ph4" "breakAfter"
    movel(ph4, a=1.2, v=0.25)
    $ 350 "MoveL"
    $ 351 "Direction: Base Z+"
    global move_thread_flag_351=0
    thread move_thread_351():
      enter_critical
      move_thread_flag_351 = 1
      local towardsPos=calculate_point_to_move_towards(p[0.0,0.0,0.0,0.0,0.0,0.0], [0.0,0.0,1.0], 1000.0)
      movel(towardsPos, a=0.1, v=0.02)
      move_thread_flag_351 = 2
      exit_critical
    end
    move_thread_flag_351 = 0
    move_thread_han_351 = run move_thread_351()
    while (True):
      local targetTcpDirection=get_target_tcp_speed()
      local stepsToRetract=tool_contact(direction=targetTcpDirection)
      if (stepsToRetract > 0):
        kill move_thread_han_351
        stopl(3.0)
        local backTrackMovement=get_actual_joint_positions_history(stepsToRetract)
        local contactPose=get_forward_kin(backTrackMovement)
        local posDir=[targetTcpDirection[0],targetTcpDirection[1],targetTcpDirection[2]]
        local retractTo=contactPose
        if (norm(posDir) > 1e-6):
          local normalizedPosDir=normalize(posDir)
          local additionalRetraction=p[normalizedPosDir[0] * 0.0, normalizedPosDir[1] * 0.0, normalizedPosDir[2] * 0.0, 0, 0, 0]
          retractTo = pose_sub(contactPose, additionalRetraction)
        end
        movel(retractTo, a=3.0, v=0.1)
        $ 352 "Until (tool_contact_detection)"
        break
      end
      sync()
    end
    $ 353 "p22≔get_actual_tcp_pose()"
    global p22= get_actual_tcp_pose ()
    $ 354 "MoveL"
    $ 355 "ph4" "breakAfter"
    movel(ph4, a=1.2, v=0.25)
    $ 356 "ph4a" "breakAfter"
    movel(ph4a, a=1.2, v=0.25)
    $ 357 "MoveJ"
    $ 358 "Waypoint_16" "breakAfter"
    movej(get_inverse_kin(Waypoint_16_p, qnear=Waypoint_16_q), a=1.3962634015954636, v=1.0471975511965976)
    $ 366 "Home"
    movej([-3.266929759358355, -1.2139462677784536, 1.5878387874396154, 1.1069165929565088, -0.0023738326664366483, -1.7891447305770605], a=1.3962634015954636, v=1.0471975511965976)
  end
  $ 2 "BeforeStart"
  $ 3 "Safe Home Folder"
  $ 4 "'if robot is not at home, send it back to home safely'"
  # 'if robot is not at home, send it back to home safely'
  $ 5 "'make sure the tcp is welder'"
  # 'make sure the tcp is welder'
  $ 6 "Set"
  set_tcp(p[-0.0095,-0.328,0.10573,1.2092,-1.2092,1.2092])
  $ 7 "sp≔get_actual_tcp_pose()"
  global sp= get_actual_tcp_pose ()
  $ 8 "MoveL"
  $ 9 "sp" "breakAfter"
  movel(sp, a=1.2, v=0.25)
  $ 10 "'if first move is to a variable, skip automove'"
  # 'if first move is to a variable, skip automove'
  $ 11 "'turn off welder'"
  # 'turn off welder'
  # begin: URCap Program Node
  #   Source: WireTank Serial, 4.9.0, WireTank, LLC
  #   Type: WireTank Serial
  $ 12 "Serial Bridge uR0"
  SerialResponse = WTSerialBridge.send_command("/dev/ttyUSB0",1200, 8, "None", "One", "None", 1000, "None", "None", [252,82,48], False)
  # end: URCap Program Node
  $ 13 "Set DO[0]=Off"
  set_standard_digital_out(0, False)
  $ 14 "jp≔get_actual_joint_positions()"
  global jp= get_actual_joint_positions ()
  $ 15 "If sp[0]>0.600"
  if (sp[0]>0.600):
    $ 16 "'if x > 600 then above then home'"
    # 'if x > 600 then above then home'
    $ 17 "MoveJ"
    $ 19 "Waypoint_76" "breakAfter"
    movej(get_inverse_kin(Waypoint_76_p, qnear=Waypoint_76_q), a=1.3962634015954636, v=1.0471975511965976)
    $ 20 "Home"
    movej([-3.266929759358355, -1.2139462677784536, 1.5878387874396154, 1.1069165929565088, -0.0023738326664366483, -1.7891447305770605], a=1.3962634015954636, v=1.0471975511965976)
  else:
    $ 21 "Else" "noBreak"
    $ 22 "Popup: retreating to home"
    popup("retreating to home", "Message", False, False, blocking=True)
    $ 23 "'for rules 2-8, finish with oldhome then above then home'"
    # 'for rules 2-8, finish with oldhome then above then home'
    $ 24 "If -1.74<jp[4] and jp[4]<1.05 and -1.74<jp[3] and jp[3]<1.74"
    if (-1.74<jp[4]  and  jp[4]<1.05  and  -1.74<jp[3]  and  jp[3]<1.74):
      $ 25 "'if oldhome, test teach, then go straight to oldhome'"
      # 'if oldhome, test teach, then go straight to oldhome'
    else:
      $ 26 "ElseIf sp[0]<-.5 and jp[3]>3.14 and -2.62<jp[4] and jp[4]<-0.87"
      if (sp[0]<-.5  and  jp[3]>3.14  and  -2.62<jp[4]  and  jp[4]<-0.87):
        $ 27 "'if left side weld approach, left weld approach in reverse'"
        # 'if left side weld approach, left weld approach in reverse'
        $ 28 "MoveJ"
        $ 29 "Waypoint_50" "breakAfter"
        movej(get_inverse_kin(Waypoint_50_p, qnear=Waypoint_50_q), a=1.3962634015954636, v=1.0471975511965976)
        $ 30 "Waypoint_51" "breakAfter"
        movej(get_inverse_kin(Waypoint_51_p, qnear=Waypoint_51_q), a=1.3962634015954636, v=1.0471975511965976)
        $ 31 "Waypoint_52" "breakAfter"
        movej(get_inverse_kin(Waypoint_52_p, qnear=Waypoint_52_q), a=1.3962634015954636, v=1.0471975511965976)
        $ 32 "Waypoint_53" "breakAfter"
        movej(get_inverse_kin(Waypoint_53_p, qnear=Waypoint_53_q), a=1.3962634015954636, v=1.0471975511965976)
      else:
        $ 33 "ElseIf sp[0]<0 and 0<jp[3] and jp[3]<1.74 and 0.87<jp[4] and jp[4]<2.62"
        if (sp[0]<0  and  0<jp[3]  and  jp[3]<1.74  and  0.87<jp[4]  and  jp[4]<2.62):
          $ 34 "'if right side around, move back then wapoint 24 then oldhome'"
          # 'if right side around, move back then wapoint 24 then oldhome'
          $ 35 "If sp[0]<-1.0"
          if (sp[0]<-1.0):
            $ 36 "xback≔p[-1.0,sp[1],sp[2],sp[3],sp[4],sp[5]]"
            global xback=p[-1.0,sp[1],sp[2],sp[3],sp[4],sp[5]]
            $ 37 "MoveJ"
            $ 38 "xback" "breakAfter"
            movej(xback, a=1.3962634015954636, v=1.0471975511965976)
          end
          $ 39 "MoveJ"
          $ 40 "Waypoint_54" "breakAfter"
          movej(get_inverse_kin(Waypoint_54_p, qnear=Waypoint_54_q), a=1.3962634015954636, v=1.0471975511965976)
        else:
          $ 41 "ElseIf jp[3]>2.62 and jp[4]<-3.84"
          if (jp[3]>2.62  and  jp[4]<-3.84):
            $ 42 "'if left side second half, then left weld ending sequence'"
            # 'if left side second half, then left weld ending sequence'
            $ 43 "If jp[5]<0.35"
            if (jp[5]<0.35):
              $ 44 "MoveJ"
              $ 45 "Waypoint_65" "breakAfter"
              movej(get_inverse_kin(Waypoint_65_p, qnear=Waypoint_65_q), a=1.3962634015954636, v=1.0471975511965976)
            end
            $ 46 "MoveJ"
            $ 51 "'above is testing, below is real'"
            # 'above is testing, below is real'
            $ 52 "Waypoint_55" "breakAfter"
            movej(get_inverse_kin(Waypoint_55_p, qnear=Waypoint_55_q), a=1.3962634015954636, v=1.0471975511965976)
            $ 54 "Waypoint_59" "breakAfter"
            movej(get_inverse_kin(Waypoint_59_p, qnear=Waypoint_59_q), t=2.0)
            $ 55 "Waypoint_71" "breakAfter"
            movej(get_inverse_kin(Waypoint_71_p, qnear=Waypoint_71_q), a=1.3962634015954636, v=1.0471975511965976)
            $ 56 "Waypoint_58" "breakAfter"
            movej(get_inverse_kin(Waypoint_58_p, qnear=Waypoint_58_q), a=1.3962634015954636, v=1.0471975511965976)
            $ 57 "Waypoint_56" "breakAfter"
            movej(get_inverse_kin(Waypoint_56_p, qnear=Waypoint_56_q), a=1.3962634015954636, v=1.0471975511965976)
            $ 58 "Waypoint_57" "breakAfter"
            movej(get_inverse_kin(Waypoint_57_p, qnear=Waypoint_57_q), a=1.3962634015954636, v=1.0471975511965976)
          else:
            $ 59 "ElseIf jp[3]<-2.09"
            if (jp[3]<-2.09):
              $ 60 "'bottom homing'"
              # 'bottom homing'
              $ 61 "MoveJ"
              $ 63 "Comment"
              # Comment
              $ 64 "If sp[0]<-0.95"
              if (sp[0]<-0.95):
                $ 65 "xback≔p[-0.95,sp[1],sp[2],sp[3],sp[4],sp[5]]"
                global xback=p[-0.95,sp[1],sp[2],sp[3],sp[4],sp[5]]
                $ 66 "MoveL"
                $ 67 "xback" "breakAfter"
                movel(xback, a=1.2, v=0.25)
              end
              $ 68 "Waypoint_67" "breakAfter"
              movej(get_inverse_kin(Waypoint_67_p, qnear=Waypoint_67_q), a=1.3962634015954636, v=1.0471975511965976)
            else:
              $ 69 "ElseIf jp[3]<0 and jp[4]<-3.14"
              if (jp[3]<0  and  jp[4]<-3.14):
                $ 70 "'if left side homing, special unspin'"
                # 'if left side homing, special unspin'
                $ 71 "MoveJ"
                $ 73 "Comment"
                # Comment
                $ 74 "Waypoint_69" "breakAfter"
                movej(get_inverse_kin(Waypoint_69_p, qnear=Waypoint_69_q), a=1.3962634015954636, v=1.0471975511965976)
                $ 75 "Waypoint_70" "breakAfter"
                movej(get_inverse_kin(Waypoint_70_p, qnear=Waypoint_70_q), a=1.3962634015954636, v=1.0471975511965976)
              else:
                $ 76 "ElseIf (sp[4]<-3 or sp[4]>3) and -0.02<sp[5] and sp[5]<0.02"
                if ((sp[4]<-3  or  sp[4]>3)  and  -0.02<sp[5]  and  sp[5]<0.02):
                  $ 77 "'go straight to home'"
                  # 'go straight to home'
                else:
                  $ 78 "ElseIf 2>1"
                  if (2>1):
                    $ 79 "'if none of the other options, then error continuously'"
                    # 'if none of the other options, then error continuously'
                    $ 80 "Loop 2>1"
                    while (2>1):
                      $ 81 "Popup: Unknown Position. Find Calvin for Assistance"
                      popup("Unknown Position. Find Calvin for Assistance", "Message", False, False, blocking=True)
                    end
                  end
                end
              end
            end
          end
        end
      end
    end
    $ 82 "'insert logic for how to get back to oldhome'"
    # 'insert logic for how to get back to oldhome'
    $ 83 "'finish with oldhome then above then home'"
    # 'finish with oldhome then above then home'
    $ 84 "MoveJ"
    $ 85 "Waypoint_49" "breakAfter"
    movej(get_inverse_kin(Waypoint_49_p, qnear=Waypoint_49_q), a=1.3962634015954636, v=1.0471975511965976)
    $ 87 "Waypoint_75" "breakAfter"
    movej(get_inverse_kin(Waypoint_75_p, qnear=Waypoint_75_q), a=1.3962634015954636, v=1.0471975511965976)
    $ 88 "Home"
    movej([-3.266929759358355, -1.2139462677784536, 1.5878387874396154, 1.1069165929565088, -0.0023738326664366483, -1.7891447305770605], a=1.3962634015954636, v=1.0471975511965976)
  end
  # begin: URCap Program Node
  #   Source: MachineLogic for Universal Robots, 3.1.7, Vention Inc.
  #   Type: MachineLogic for Universal Robots
  $ 89 "MachineLogic Homing"
  while isVentionMovementBusyMachineMotion1==True:
  sleep(0.05)
  end
  if(isVentionMovementBusyMachineMotion1 == False):
  isVentionMovementBusyMachineMotion1 = True
  socket_send_string("estop/status;", "MachineMotion1")
  temp_estop_var_vention = socket_read_string("MachineMotion1",timeout=15)
  while(temp_estop_var_vention=="estop/status true"):
  if temp_estop_var_vention=="estop/status true":
  sendStringWithTimeout("estop/systemreset/request","Ack estop/systemreset/request;","MachineMotion1")
  end
  socket_send_string("estop/status;", "MachineMotion1")
  temp_estop_var_vention = socket_read_string("MachineMotion1",timeout=15)
  if temp_estop_var_vention=="estop/status true":
  popup("MachineMotion in estop, make sure you have all emergency modules released manually. If you continue the system will try to reset MachineMotion automatically.",blocking=True)
  end
  end
  else:
  popup("resource is being used already: MachineMotion1")
  halt
  end
  isVentionMovementBusyMachineMotion1 = True
  sendString("im_home_axis_1", "MachineMotion im_home_axis_1 = completed", "MachineMotion1")
  isVentionMovementBusyMachineMotion1 = False
  sendString("SET im_set_encoder_pos_aux_1 0.000", "Ack", "MachineMotion1")
  isVentionMovementBusyMachineMotion1 = False
  sleep(0.03)
  # end: URCap Program Node
  $ 367 "Thread_1"
  thread Thread_1():
    $ 368 "Loop  True "
    while (  True  ):
      $ 369 "If freedrive_m_var≟ True "
      if (freedrive_m_var ==   True  ):
        $ 370 "freedrive_mode()"
        freedrive_mode()
        $ 371 "free_dr_already≔ True "
        global free_dr_already=  True
      else:
        $ 372 "Else" "noBreak"
        $ 373 "If free_dr_already"
        if (free_dr_already):
          $ 374 "end_freedrive_mode()"
          end_freedrive_mode()
        end
      end
      $ 375 "sync()"
      sync()
    end
  end
  threadId_Thread_1 = run Thread_1()
  $ 90 "Robot Program"
  $ 91 "'start of main program'"
  # 'start of main program'
  $ 92 "Set"
  set_tcp(p[-0.0095,-0.328,0.10573,1.2092,-1.2092,1.2092])
  $ 93 "Home"
  movej([-3.266929759358355, -1.2139462677784536, 1.5878387874396154, 1.1069165929565088, -0.0023738326664366483, -1.7891447305770605], a=1.3962634015954636, v=1.0471975511965976)
  $ 94 "Script: analyze_touchpoints.script"
  # this file creates the function for analyzing touchpoints
  # define pi
  pi = 3.1415926535
  # initialize a lift column extension needed of 0.0
  global liftcolumnzneeded = 0.0

  # this is the main entry point for calculations.
  # it takes in the 5 points, analyzes the shape of the box, and then calculates path points and returns them
  # specifically for Down, Over, then Around (DOtA)
  # specifically for right-sided boxes (vertical weld on right side of edge)
  def main_calculate_right(p11, p12, p21, p22, p3, p13, p23, chamferover):
      struct1 = analyze_touchpoints_only(p11, p12, p21, p22, p3)
      list1 = analyze_vertical_touchpoints(p11, p12, p13, p21, p22, p23, p3)
      struct2 = calculate_DOtA_points_right(struct1, list1, chamferover)
      validity = check_validity_right(struct1, struct2)
      return struct2
  end

  # this is the main entry point for calculations.
  # it takes in the 5 points, analyzes the shape of the box, and then calculates path points and returns them
  # specifically for Down, Over, then Around (DOtA)
  # specifically for left-sided boxes (vertical weld on left side of edge)
  def main_calculate_left(p11, p12, p21, p22, p3, p13, p23, chamferover):
      struct1 = analyze_touchpoints_only(p11, p12, p21, p22, p3)
      list1 = analyze_vertical_touchpoints(p11, p12, p13, p21, p22, p23, p3)
      struct2 = calculate_DOtA_points_left(struct1, list1, chamferover)
      validity = check_validity_left(struct1, struct2)
      return struct2
  end

  # this is the main entry point for calculations, for Floor Corner Extended.
  # it takes in the 7 touchpoints, analyzes the shape of the box.
  # takes in the user defined point for the top of the weld (tcp_pose_top) and then calculates path points
  # loopingly tries to calculate the extension along the sidewall that fulfills get_inverse_kin_has_solution() and provides the farthest extension possible
  # returns the pathpoints
  # specifically for Down, Over, then Around (DOtA)
  # specifically for right-sided boxes (vertical weld on right side of edge)
  def main_calculate_right_extended(p11, p12, p21, p22, p3, p13, p23, chamferover, chamferup, tcp_pose_top):
      struct1 = analyze_touchpoints_only(p11, p12, p21, p22, p3)
      list1 = analyze_vertical_touchpoints(p11, p12, p13, p21, p22, p23, p3)
      struct2 = calculate_DOtA_points_right_extended(struct1, list1, chamferover, chamferup, tcp_pose_top)
      struct3 = check_validity_right(struct1, struct2)
      return struct3
  end

  # this is the main entry point for calculations, for Floor Corner Extended.
  # it takes in the 7 touchpoints, analyzes the shape of the box.
  # takes in the user defined point for the top of the weld (tcp_pose_top) and then calculates path points
  # loopingly tries to calculate the extension along the sidewall that fulfills get_inverse_kin_has_solution() and provides the farthest extension possible
  # returns the pathpoints
  # specifically for Down, Over, then Around (DOtA)
  # specifically for left-sided boxes (vertical weld on left side of edge)
  def main_calculate_left_extended(p11, p12, p21, p22, p3, p13, p23, chamferover, chamferup, tcp_pose_top):
      struct1 = analyze_touchpoints_only(p11, p12, p21, p22, p3)
      list1 = analyze_vertical_touchpoints(p11, p12, p13, p21, p22, p23, p3)
      struct2 = calculate_DOtA_points_left_extended(struct1, list1, chamferover, chamferup, tcp_pose_top)
      struct3 = check_validity_left(struct1, struct2)
      return struct3
  end

  # it takes 5 arguments as points
  # it returns a struct containing: (pointintersect, pointapproach1, pointapproach2, point1, point2, point3, point4, point5, pointreturn1, heading1, heading2, heading3, path2r1, path2r2, path2l1, path2l2)
  # specifically for Around then Up (AtU)
  def analyze_touchpoints(p11, p12, p21, p22, p3):
    # FIND THE INTERSECTION
    # comment get the z
    zcoord=p3[2]

    # get the raw points from the first line
    l1p1x=p11[0]
    l1p1y=p11[1]
    l1p2x=p12[0]
    l1p2y=p12[1]

    # equate the first line in 2d space
    ml1 = (l1p2y-l1p1y) / (l1p2x-l1p1x)

    # b = y - mx
    bl1 = l1p1y - ml1 * l1p1x

    # get the raw points from the second line
    l2p1x=p21[0]
    l2p1y=p21[1]
    l2p2x=p22[0]
    l2p2y=p22[1]

    # equate the second line in 2d space
    ml2 = (l2p2y-l2p1y) / (l2p2x-l2p1x)

    # b = y - mx
    bl2 = l2p1y - ml2 * l2p1x


    # find the intersection of the two lines
    # m1x+b1 = m2x+b2
    # m1x - m2x = b2 - b1
    # x = (b2-b1) / (m1-m2)
    xintersect = (bl2-bl1) / (ml1-ml2)
    yintersect = ml1 * xintersect + bl1

    #FIND THE VECTORS
    #define a vector from the intersection to the second point on the first line
    l1delxfull = l1p2x - xintersect
    l1delyfull = l1p2y - yintersect

    l1delmag = sqrt(l1delxfull*l1delxfull + l1delyfull*l1delyfull)

    l1delxunit = l1delxfull / l1delmag
    l1delyunit = l1delyfull / l1delmag

    #define a vector from the intersection to the second point on the second line
    l2delxfull = l2p2x - xintersect
    l2delyfull = l2p2y - yintersect

    l2delmag = sqrt(l2delxfull*l2delxfull + l2delyfull*l2delyfull)

    l2delxunit = l2delxfull / l2delmag
    l2delyunit = l2delyfull / l2delmag

    # FIND THE FOUR POINTS ON THE LINES
    # find locations 8 inches away from  intersect point
    # CONST
    welddistance = 8
    roundoverdistance = 0.05
    zup = .375
    # inches
    wd = welddistance * 25.4 / 1000
    rod = roundoverdistance * 25.4 / 1000
    zup = zup * 25.4 / 1000

    # now we have the unit vector. extend the weld distance from the intersection
    x = xintersect + l1delxunit * wd
    y = yintersect + l1delyunit * wd
    z = zcoord + zup

    point1 = p[x,y,z,1.570796,0,0] # dummy orientation for now

    x = xintersect + l1delxunit * rod
    y = yintersect + l1delyunit * rod

    point2 = p[x,y,z,1.570796,0,0]

    # now we have the unit vector. extend the weld distance from the intersection
    x = xintersect + l2delxunit * wd
    y = yintersect + l2delyunit * wd

    point5 = p[x,y,z,0,-1.570796,0]

    x = xintersect + l2delxunit * rod
    y = yintersect + l2delyunit * rod

    point4 = p[x,y,z,0,-1.570796,0]

    #DEFINE APPROACH POINTS
    pointintersect = p[xintersect,yintersect,zcoord,0,0,0]
    pointapproach1 = p[xintersect+0.1,yintersect+0.1,z,1.570796,0,0]
    pointapproach2 = p[point1[0], point1[1]+0.1, point1[2], point1[3], point1[4], point1[5]]
    pointreturn1 = p[point5[0]+0.1, point5[1], point5[2], point5[3], point5[4], point5[5]]

    #FIND HEADINGS
    #for each heading, find the angle of the line with respect to the pos x axis. then add/subtract 90 degrees because you want to be perpendicular to that
    headingvector1 = convert_uv_to_heading(l1delxunit, l1delyunit)
    headingvector2 = convert_uv_to_heading(l2delxunit, l2delyunit)
    # find halfway heading
    heading2 = (headingvector1 + headingvector2)/2
    # find headings that the robot should face while traveling, perpendicular to the vectors of the sides of the box
    heading1 = headingvector1 + pi/2
    heading3 = headingvector2 - pi/2

    #FIND POINT 3
    #see if we have to / can find point 3
    findpoint3 = True
    if roundoverdistance == 0:
      findpoint3 = False
    end
    if findpoint3:
      # i need to find the point3 such that the arc from p2 to p3 to p4 is tangent to p1-p2 and p4-p5. making this a smooth path will be good
      # the direction of movement is from pointintersect in the direction of heading2
      # how much movement though? this will depend on whether it is actually a 90 degree angle or not.
      # first, find the perpendicular lines through points 2 and 4
      perp2 = find_perpendicular_line(ml1, point2[0], point2[1])
      perp4 = find_perpendicular_line(ml2, point4[0], point4[1])
      # next, find the intersection of those two lines
      perpintersect = find_intersection(perp2[0], perp2[1], perp4[0], perp4[1])
      radiusofcircle = distance_between(perpintersect[0], perpintersect[1], 0, point2[0], point2[1], 0)
      # find a vector the direction of heading2
      uvx = cos(heading2)
      uvy = sin(heading2)
      # compute point3. pass in negative radius because the direction is into the tank but we want to move from the intersection out to the rounded edge
      point3coords = add_vectordistance_to_point(perpintersect[0], perpintersect[1], z, uvx, uvy, 0, -1 * radiusofcircle)
      point3 = p[point3coords[0], point3coords[1], point3coords[2], 0, 0, 0]
    end

    #APPLY ACTUAL RXRYRZ TO POINTS
    # convert the headings to rxryrz and insert those values into the relevant points
    rxryrz = convert_heading_to_axang(heading1)
    rx = rxryrz[0]
    ry = rxryrz[1]
    rz = rxryrz[2]
    pointapproach1 = p[pointapproach1[0], pointapproach1[1], pointapproach1[2], rx, ry, rz]
    pointapproach2 = p[pointapproach2[0], pointapproach2[1], pointapproach2[2], rx, ry, rz]
    point1 = p[point1[0], point1[1], point1[2], rx, ry, rz]
    point2 = p[point2[0], point2[1], point2[2], rx, ry, rz]
    rxryrz = convert_heading_to_axang(heading2)
    rx = rxryrz[0]
    ry = rxryrz[1]
    rz = rxryrz[2]
    if findpoint3:
      point3 = p[point3[0], point3[1], point3[2], rx, ry, rz]
    else:
      point3 = point2
    end
    rxryrz = convert_heading_to_axang(heading3)
    rx = rxryrz[0]
    ry = rxryrz[1]
    rz = rxryrz[2]
    point4 = p[point4[0], point4[1], point4[2], rx, ry, rz]
    point5 = p[point5[0], point5[1], point5[2], rx, ry, rz]
    pointreturn1 = p[pointreturn1[0], pointreturn1[1], pointreturn1[2], rx, ry, rz]

    #find path2 (the part that goes up)
    four_vertical_points = find_vertical_points(pointintersect, l1delxunit, l1delyunit, l2delxunit, l2delyunit, zup, wd, heading1, heading3)
    path2r1 = four_vertical_points[0]
    path2r2 = four_vertical_points[1]
    path2l1 = four_vertical_points[2]
    path2l2 = four_vertical_points[3]

    #RETURN STRUCT
    ret = struct(pointintersect=pointintersect, pointapproach1=pointapproach1, pointapproach2=pointapproach2, point1=point1, point2=point2, point3=point3, point4=point4, point5=point5, pointreturn1=pointreturn1, heading1=heading1, heading2=heading2, heading3=heading3, path2r1=path2r1, path2r2=path2r2, path2l1=path2l1, path2l2=path2l2)
    return ret
  end

  # based on a Corner Homing 45 Cover pattern of touchpoints
  # this uses those touchpoints to create a representation of the corner in 3d robot space.
  def analyze_touchpoints_only_cover(p11, p12, p21, p3):
      zcoord=p3[2]

      # get the raw points from the first line
      l1p1x=p11[0]
      l1p1y=p11[1]
      l1p2x=p12[0]
      l1p2y=p12[1]

      # equate the first line in 2d space
      ml1 = (l1p2y-l1p1y) / (l1p2x-l1p1x)

      # b = y - mx
      bl1 = l1p1y - ml1 * l1p1x

      # get the raw points from the second line
      l2p1x=p21[0]
      l2p1y=p21[1]

      # equate the second line in 2d space
      # ml2 = opposite reciprocal of ml1 (because they are perpendicular) (assume perpendicular to make calculation of weldpath much easier)
      ml2 = -1 / ml1

      # b = y - mx
      bl2 = l2p1y - ml2 * l2p1x

      # find the intersection of the two lines
      # m1x+b1 = m2x+b2
      # m1x - m2x = b2 - b1
      # x = (b2-b1) / (m1-m2)
      xintersect = (bl2-bl1) / (ml1-ml2)
      yintersect = ml1 * xintersect + bl1

      pointintersect = p[xintersect,yintersect,zcoord,0,0,0]

      #FIND THE VECTORS
      #define a vector from the intersection to the second point on the first line
      l1delxfull = l1p2x - xintersect
      l1delyfull = l1p2y - yintersect

      l1delmag = sqrt(l1delxfull*l1delxfull + l1delyfull*l1delyfull)

      l1delxunit = l1delxfull / l1delmag
      l1delyunit = l1delyfull / l1delmag

      #define a vector from the intersection to the second point on the second line
      l2delxfull = l2p1x - xintersect
      l2delyfull = l2p1y - yintersect

      l2delmag = sqrt(l2delxfull*l2delxfull + l2delyfull*l2delyfull)

      l2delxunit = l2delxfull / l2delmag
      l2delyunit = l2delyfull / l2delmag

      #FIND HEADINGS
      #for each heading, find the angle of the line with respect to the pos x axis. this line is from pointintersect and along each edge of the corner
      heading1 = convert_uv_to_heading(l1delxunit, l1delyunit)
      heading3 = convert_uv_to_heading(l2delxunit, l2delyunit)
      # find halfway heading
      heading2 = (heading1 + heading3)/2

      #RETURN STRUCT
      ret = struct(pointintersect=pointintersect, heading1=heading1, heading2=heading2, heading3=heading3, l1delxunit=l1delxunit, l1delyunit=l1delyunit, l2delxunit=l2delxunit, l2delyunit=l2delyunit)
      return ret
  end

  # it takes 5 arguments as points
  # it returns a struct containing: (pointintersect, heading1, heading2, heading3, l1delxunit, l1delyunit, l2delxunit, l2delyunit)
  def analyze_touchpoints_only(p11, p12, p21, p22, p3):
    # FIND THE INTERSECTION
    # comment get the z
    zcoord=p3[2]

    # get the raw points from the first line
    l1p1x=p11[0]
    l1p1y=p11[1]
    l1p2x=p12[0]
    l1p2y=p12[1]

    # equate the first line in 2d space
    ml1 = (l1p2y-l1p1y) / (l1p2x-l1p1x)

    # b = y - mx
    bl1 = l1p1y - ml1 * l1p1x

    # get the raw points from the second line
    l2p1x=p21[0]
    l2p1y=p21[1]
    l2p2x=p22[0]
    l2p2y=p22[1]

    # equate the second line in 2d space
    ml2 = (l2p2y-l2p1y) / (l2p2x-l2p1x)

    # b = y - mx
    bl2 = l2p1y - ml2 * l2p1x


    # find the intersection of the two lines
    # m1x+b1 = m2x+b2
    # m1x - m2x = b2 - b1
    # x = (b2-b1) / (m1-m2)
    xintersect = (bl2-bl1) / (ml1-ml2)
    yintersect = ml1 * xintersect + bl1

    pointintersect = p[xintersect,yintersect,zcoord,0,0,0]

    #FIND THE VECTORS
    #define a vector from the intersection to the second point on the first line
    l1delxfull = l1p2x - xintersect
    l1delyfull = l1p2y - yintersect

    l1delmag = sqrt(l1delxfull*l1delxfull + l1delyfull*l1delyfull)

    l1delxunit = l1delxfull / l1delmag
    l1delyunit = l1delyfull / l1delmag

    #define a vector from the intersection to the second point on the second line
    l2delxfull = l2p2x - xintersect
    l2delyfull = l2p2y - yintersect

    l2delmag = sqrt(l2delxfull*l2delxfull + l2delyfull*l2delyfull)

    l2delxunit = l2delxfull / l2delmag
    l2delyunit = l2delyfull / l2delmag

    #FIND HEADINGS
    #for each heading, find the angle of the line with respect to the pos x axis. then add/subtract 90 degrees because you want to be perpendicular to that
    headingvector1 = convert_uv_to_heading(l1delxunit, l1delyunit)
    headingvector2 = convert_uv_to_heading(l2delxunit, l2delyunit)
    # find halfway heading
    heading2 = (headingvector1 + headingvector2)/2
    # find headings that the robot should face while traveling, perpendicular to the vectors of the sides of the box
    heading1 = headingvector1 + pi/2
    heading3 = headingvector2 - pi/2

    #RETURN STRUCT
    ret = struct(pointintersect=pointintersect, heading1=heading1, heading2=heading2, heading3=heading3, l1delxunit=l1delxunit, l1delyunit=l1delyunit, l2delxunit=l2delxunit, l2delyunit=l2delyunit)
    return ret
  end

  # given a struct from analyze_touchpoints_only(), calculate the points
  # for right, for non-extended
  def calculate_DOtA_points_right(struct1, listleans, chamferover):
      # get the stuff from the struct
      pointintersect = struct1[0]
      heading1 = struct1[1]
      heading2 = struct1[2]
      heading3 = struct1[3]
      l1delxunit = struct1[4]
      l1delyunit = struct1[5]
      l2delxunit = struct1[6]
      l2delyunit = struct1[7]

      # FIND THE POINTS ON THE LINES OF THE FIRST TURN PATH
      # find locations 8 inches away from  intersect point
      # CONST
      welddistance1 = 8 # vertical weld distance
      welddistance2 = 6 # first path second leg
      welddistance3 = 8 # second path second leg
      zup = .375
      # inches
      wd1 = welddistance1 * 25.4 / 1000
      wd2 = welddistance2 * 25.4 / 1000
      wd3 = welddistance3 * 25.4 / 1000
      zup = zup * 25.4 / 1000
      chamferovermm =  chamferover * 25.4 / 1000

      x = pointintersect[0] + l1delxunit * chamferovermm
      y = pointintersect[1] + l1delyunit * chamferovermm
      z = pointintersect[2] + zup

      #apply actual rxryrz to points
      # convert the headings to rxryrz and insert those values into the relevant points
      rxryrz = convert_heading_to_axang_preheatdown(heading1)
      rx = rxryrz[0]
      ry = rxryrz[1]
      rz = rxryrz[2]

      point1 = p[x + wd1*listleans[0], y + wd1*listleans[1], z + wd1, rx, ry, rz] # add in the listleans factor to follow the face of the box as we move up
      point2 = p[x, y, z, rx, ry, rz]

      # convert the headings to rxryrz and insert those values into the relevant points
      rxryrz = convert_heading_to_axang_ccw(heading1)
      rx = rxryrz[0]
      ry = rxryrz[1]
      rz = rxryrz[2]

      point4 = p[x, y, z, rx, ry, rz]
      x = x + l1delxunit * wd2
      y = y + l1delyunit * wd2
      point5 = p[x, y, z, rx, ry, rz]

      # FIND THE POINTS ON THE LINES OF THE SECOND AROUND PATH
      roundoverdistance = 0.05
      rod = roundoverdistance * 25.4 / 1000

      # now we have the unit vector. extend the weld distance from the intersection
      x = pointintersect[0] + l1delxunit * chamferovermm
      y = pointintersect[1] + l1delyunit * chamferovermm
      # convert the headings to rxryrz and insert those values into the relevant points
      rxryrz = convert_heading_to_axang(heading1)
      rx = rxryrz[0]
      ry = rxryrz[1]
      rz = rxryrz[2]
      point_1 = p[x, y, z, rx, ry, rz]

      x = pointintersect[0] + l1delxunit * rod
      y = pointintersect[1] + l1delyunit * rod
      point_2 = p[x, y, z, rx, ry, rz]

      # now we have the unit vector. extend the weld distance from the intersection
      x = pointintersect[0] + l2delxunit * wd3
      y = pointintersect[1] + l2delyunit * wd3
      # convert the headings to rxryrz and insert those values into the relevant points
      rxryrz = convert_heading_to_axang(heading3)
      rx = rxryrz[0]
      ry = rxryrz[1]
      rz = rxryrz[2]
      point_5 = p[x, y, z, rx, ry, rz]

      x = pointintersect[0] + l2delxunit * rod
      y = pointintersect[1] + l2delyunit * rod
      point_4 = p[x, y, z, rx, ry, rz]

      #FIND POINT 3
      # by calling analyze_touchpoints()
      atret = analyze_touchpoints(point_2, point_1, point_4, point_5, pointintersect)
      point_3 = atret[5]


      struct2 = struct(point1=point1, point2=point2, point4=point4, point5=point5, point_1=point_1, point_2=point_2, point_3=point_3, point_4=point_4, point_5=point_5)
      return struct2
  end

  # given a struct from analyze_touchpoints_only(), calculate the points
  # for left, for non-extended
  def calculate_DOtA_points_left(struct1, listleans, chamferover):
      # get the stuff from the struct
      pointintersect = struct1[0]
      heading1 = struct1[1]
      heading2 = struct1[2]
      heading3 = struct1[3]
      l1delxunit = struct1[4]
      l1delyunit = struct1[5]
      l2delxunit = struct1[6]
      l2delyunit = struct1[7]

      # FIND THE POINTS ON THE LINES OF THE FIRST TURN PATH
      # find locations 8 inches away from  intersect point
      # CONST
      welddistance1 = 8 # vertical weld distance
      welddistance2 = 6 # first path second leg
      welddistance3 = 8 # second path second leg
      zup = .375
      # inches
      wd1 = welddistance1 * 25.4 / 1000
      wd2 = welddistance2 * 25.4 / 1000
      wd3 = welddistance3 * 25.4 / 1000
      zup = zup * 25.4 / 1000
      chamferovermm =  chamferover * 25.4 / 1000

      x = pointintersect[0] + l2delxunit * chamferovermm
      y = pointintersect[1] + l2delyunit * chamferovermm
      z = pointintersect[2] + zup

      #apply actual rxryrz to points
      # convert the headings to rxryrz and insert those values into the relevant points
      rxryrz = convert_heading_to_axang_preheatdown(heading3)
      rx = rxryrz[0]
      ry = rxryrz[1]
      rz = rxryrz[2]

      point1 = p[x + wd1*listleans[0], y + wd1*listleans[1], z + wd1, rx, ry, rz]
      point2 = p[x, y, z, rx, ry, rz]

      # convert the headings to rxryrz and insert those values into the relevant points
      rxryrz = convert_heading_to_axang(heading3)
      rx = rxryrz[0]
      ry = rxryrz[1]
      rz = rxryrz[2]

      point4 = p[x, y, z, rx, ry, rz]
      x = x + l2delxunit * wd2
      y = y + l2delyunit * wd2
      point5 = p[x, y, z, rx, ry, rz]

      # FIND THE POINTS ON THE LINES OF THE SECOND AROUND PATH
      roundoverdistance = 0.05
      rod = roundoverdistance * 25.4 / 1000

      # now we have the unit vector. extend the weld distance from the intersection
      x = pointintersect[0] + l2delxunit * chamferovermm
      y = pointintersect[1] + l2delyunit * chamferovermm
      # convert the headings to rxryrz and insert those values into the relevant points
      rxryrz = convert_heading_to_axang_ccw(heading3)
      rx = rxryrz[0]
      ry = rxryrz[1]
      rz = rxryrz[2]
      point_1 = p[x, y, z, rx, ry, rz]

      x = pointintersect[0] + l2delxunit * rod
      y = pointintersect[1] + l2delyunit * rod
      point_2 = p[x, y, z, rx, ry, rz]

      # now we have the unit vector. extend the weld distance from the intersection
      x = pointintersect[0] + l1delxunit * wd3
      y = pointintersect[1] + l1delyunit * wd3
      # convert the headings to rxryrz and insert those values into the relevant points
      rxryrz = convert_heading_to_axang_ccw(heading1)
      rx = rxryrz[0]
      ry = rxryrz[1]
      rz = rxryrz[2]
      point_5 = p[x, y, z, rx, ry, rz]

      x = pointintersect[0] + l1delxunit * rod
      y = pointintersect[1] + l1delyunit * rod
      point_4 = p[x, y, z, rx, ry, rz]

      #FIND POINT 3
      # by calling analyze_touchpoints()
      atret = analyze_touchpoints(point_2, point_1, point_4, point_5, pointintersect)
      point_3 = atret[5]
      #point 3 will not have the correct rxryrz though because now the gun needs to be face up.
      rxryrz = convert_heading_to_axang_ccw(heading2)
      rx = rxryrz[0]
      ry = rxryrz[1]
      rz = rxryrz[2]
      point_3 = p[point_3[0], point_3[1], point_3[2], rx, ry, rz]

      struct2 = struct(point1=point1, point2=point2, point4=point4, point5=point5, point_1=point_1, point_2=point_2, point_3=point_3, point_4=point_4, point_5=point_5)
      return struct2
  end

  # given a struct from analyze_touchpoints_only(), calculate the points
  # for right, for extended
  def calculate_DOtA_points_right_extended(struct1, listleans, chamferover, chamferup, tcp_pose_top):
      # get the stuff from the struct
      pointintersect = struct1[0]
      heading1 = struct1[1]
      heading2 = struct1[2]
      heading3 = struct1[3]
      l1delxunit = struct1[4]
      l1delyunit = struct1[5]
      l2delxunit = struct1[6]
      l2delyunit = struct1[7]

      # FIND THE POINTS ON THE LINES OF THE FIRST TURN PATH
      # find locations 8 inches away from  intersect point
      # CONST
      # welddistance1 = 8 # vertical weld distance
      welddistance2 = 6 # first path second leg
      welddistance3 = 8 # second path second leg

      # inches
      # wd1 = welddistance1 * 25.4 / 1000
      wd2 = welddistance2 * 25.4 / 1000
      wd3 = welddistance3 * 25.4 / 1000
      zup = chamferup * 25.4 / 1000
      chamferovermm =  chamferover * 25.4 / 1000

      # weld distance is the distance that it will weld. this will make it start at the z height that the user specified
      wd1 = tcp_pose_top[2] - pointintersect[2] - zup

      x = pointintersect[0] + l1delxunit * chamferovermm
      y = pointintersect[1] + l1delyunit * chamferovermm
      z = pointintersect[2] + zup

      #apply actual rxryrz to points
      # convert the headings to rxryrz and insert those values into the relevant points
      rxryrz = convert_heading_to_axang_preheatdown(heading1)
      rx = rxryrz[0]
      ry = rxryrz[1]
      rz = rxryrz[2]

      point1 = p[x + wd1*listleans[0], y + wd1*listleans[1], z + wd1, rx, ry, rz] # add in the listleans factor to follow the face of the box as we move up
      point2 = p[x, y, z, rx, ry, rz]

      # convert the headings to rxryrz and insert those values into the relevant points
      rxryrz = convert_heading_to_axang_ccw(heading1)
      rx = rxryrz[0]
      ry = rxryrz[1]
      rz = rxryrz[2]

      point4 = p[x, y, z, rx, ry, rz]
      x = x + l1delxunit * wd2
      y = y + l1delyunit * wd2
      point5 = p[x, y, z, rx, ry, rz]

      # FIND THE POINTS ON THE LINES OF THE SECOND AROUND PATH
      roundoverdistance = 0.05
      rod = roundoverdistance * 25.4 / 1000

      # now we have the unit vector. extend the weld distance from the intersection
      x = pointintersect[0] + l1delxunit * chamferovermm
      y = pointintersect[1] + l1delyunit * chamferovermm
      # convert the headings to rxryrz and insert those values into the relevant points
      rxryrz = convert_heading_to_axang(heading1)
      rx = rxryrz[0]
      ry = rxryrz[1]
      rz = rxryrz[2]
      point_1 = p[x, y, z, rx, ry, rz]

      x = pointintersect[0] + l1delxunit * rod
      y = pointintersect[1] + l1delyunit * rod
      point_2 = p[x, y, z, rx, ry, rz]

      # convert the headings to rxryrz and insert those values into the relevant points
      rxryrz = convert_heading_to_axang(heading3)
      rx = rxryrz[0]
      ry = rxryrz[1]
      rz = rxryrz[2]

      x = pointintersect[0] + l2delxunit * rod
      y = pointintersect[1] + l2delyunit * rod
      point_4 = p[x, y, z, rx, ry, rz]

      # now we have the unit vector. extend the weld distance from the intersection
      x = pointintersect[0] + l2delxunit * wd3
      y = pointintersect[1] + l2delyunit * wd3
      point_5 = p[x, y, z, rx, ry, rz]

      #FIND POINT 3
      # by calling analyze_touchpoints()
      atret = analyze_touchpoints(point_2, point_1, point_4, point_5, pointintersect)
      atret5 = atret[5]
      point_3 = p[atret5[0], atret5[1], z, atret5[3], atret5[4], atret5[5]]


      struct2 = struct(point1=point1, point2=point2, point4=point4, point5=point5, point_1=point_1, point_2=point_2, point_3=point_3, point_4=point_4, point_5=point_5)
      return struct2
  end

  # given a struct from analyze_touchpoints_only(), calculate the points
  # for left, for extended
  def calculate_DOtA_points_left_extended(struct1, listleans, chamferover, chamferup, tcp_pose_top):
      # get the stuff from the struct
      pointintersect = struct1[0]
      heading1 = struct1[1]
      heading2 = struct1[2]
      heading3 = struct1[3]
      l1delxunit = struct1[4]
      l1delyunit = struct1[5]
      l2delxunit = struct1[6]
      l2delyunit = struct1[7]

      # FIND THE POINTS ON THE LINES OF THE FIRST TURN PATH
      # find locations 8 inches away from  intersect point
      # CONST
      # welddistance1 = 8 # vertical weld distance
      welddistance2 = 6 # first path second leg
      welddistance3 = 8 # second path second leg

      # inches
      # wd1 = welddistance1 * 25.4 / 1000
      wd2 = welddistance2 * 25.4 / 1000
      wd3 = welddistance3 * 25.4 / 1000
      zup = chamferup * 25.4 / 1000
      chamferovermm =  chamferover * 25.4 / 1000

      # weld distance is the distance that it will weld. this will make it start at the z height that the user specified
      wd1 = tcp_pose_top[2] - pointintersect[2] - zup

      x = pointintersect[0] + l2delxunit * chamferovermm
      y = pointintersect[1] + l2delyunit * chamferovermm
      z = pointintersect[2] + zup

      #apply actual rxryrz to points
      # convert the headings to rxryrz and insert those values into the relevant points
      rxryrz = convert_heading_to_axang_preheatdown(heading3)
      rx = rxryrz[0]
      ry = rxryrz[1]
      rz = rxryrz[2]

      point1 = p[x + wd1*listleans[0], y + wd1*listleans[1], z + wd1, rx, ry, rz]
      point2 = p[x, y, z, rx, ry, rz]

      # convert the headings to rxryrz and insert those values into the relevant points
      rxryrz = convert_heading_to_axang(heading3)
      rx = rxryrz[0]
      ry = rxryrz[1]
      rz = rxryrz[2]

      point4 = p[x, y, z, rx, ry, rz]
      x = x + l2delxunit * wd2
      y = y + l2delyunit * wd2
      point5 = p[x, y, z, rx, ry, rz]

      # FIND THE POINTS ON THE LINES OF THE SECOND AROUND PATH
      roundoverdistance = 0.05
      rod = roundoverdistance * 25.4 / 1000

      # now we have the unit vector. extend the weld distance from the intersection
      x = pointintersect[0] + l2delxunit * chamferovermm
      y = pointintersect[1] + l2delyunit * chamferovermm
      # convert the headings to rxryrz and insert those values into the relevant points
      rxryrz = convert_heading_to_axang_ccw(heading3)
      rx = rxryrz[0]
      ry = rxryrz[1]
      rz = rxryrz[2]
      point_1 = p[x, y, z, rx, ry, rz]

      x = pointintersect[0] + l2delxunit * rod
      y = pointintersect[1] + l2delyunit * rod
      point_2 = p[x, y, z, rx, ry, rz]

      # convert the headings to rxryrz and insert those values into the relevant points
      rxryrz = convert_heading_to_axang_ccw(heading1)
      rx = rxryrz[0]
      ry = rxryrz[1]
      rz = rxryrz[2]

      x = pointintersect[0] + l1delxunit * rod
      y = pointintersect[1] + l1delyunit * rod
      point_4 = p[x, y, z, rx, ry, rz]

      # now we have the unit vector. extend the weld distance from the intersection
      x = pointintersect[0] + l1delxunit * wd3
      y = pointintersect[1] + l1delyunit * wd3
      point_5 = p[x, y, z, rx, ry, rz]

      #FIND POINT 3
      # by calling analyze_touchpoints()
      atret = analyze_touchpoints(point_2, point_1, point_4, point_5, pointintersect)
      point_3 = atret[5]
      #point 3 will not have the correct rxryrz though because now the gun needs to be face up
      rxryrz = convert_heading_to_axang_ccw(heading2)
      rx = rxryrz[0]
      ry = rxryrz[1]
      rz = rxryrz[2]
      point_3 = p[point_3[0], point_3[1], z, rx, ry, rz]

      struct2 = struct(point1=point1, point2=point2, point4=point4, point5=point5, point_1=point_1, point_2=point_2, point_3=point_3, point_4=point_4, point_5=point_5)
      return struct2
  end

